	X =  1242.484  mm,	Y =   -38.517  mm,	Z =  2264.100  mm,
	W =   -32.017 deg,	P =   -31.509 deg,	R =    19.354 deg
   GP2:
	UF : 0, UT : 1,
	J1=   131.188 deg,	J2=   180.000 deg
};
P[910]{
   GP1:
	UF : 1, UT : 1,		CONFIG : 'N U T, 0, 0, 0',
	X =  1678.533  mm,	Y =  -253.828  mm,	Z =  2096.179  mm,
	W =   -44.666 deg,	P =    -5.995 deg,	R =    -2.790 deg
   GP2:
	UF : 0, UT : 1,
	J1=   131.188 deg,	J2=   180.000 deg
};
P[911]{
   GP1:
	UF : 1, UT : 1,		CONFIG : 'N U T, 0, 0, 0',
	X =  1703.320  mm,	Y =  -397.922  mm,	Z =  1954.333  mm,
	W =   -45.225 deg,	P =    -9.980 deg,	R =     1.224 deg
   GP2:
	UF : 0, UT : 1,
	J1=   131.188 deg,	J2=   180.000 deg
};
P[912]{
   GP1:
	UF : 1, UT : 1,		CONFIG : 'N U T, 0, 0, 0',
	X =  1675.864  mm,	Y =  -397.713  mm,	Z =  1947.138  mm,
	W =   -45.494 deg,	P =    11.391 deg,	R =   -20.046 deg
   GP2:
	UF : 0, UT : 1,
	J1=   131.188 deg,	J2=   180.000 deg
};
P[913]{
   GP1:
	UF : 1, UT : 1,		CONFIG : 'N U T, 0, 0, 0',
	X =  1728.670  mm,	Y =  -309.937  mm,	Z =  2044.029  mm,
	W =   -44.670 deg,	P =    -6.034 deg,	R =    -2.751 deg
   GP2:
	UF : 0, UT : 1,
	J1=   131.188 deg,	J2=   180.000 deg
};
P[914]{
   GP1:
	UF : 1, UT : 1,		CONFIG : 'N U T, 0, 0, 0',
	X =  1347.300  mm,	Y =  -220.973  mm,	Z =  2082.770  mm,
	W =    -1.262 deg,	P =   -15.279 deg,	R =     7.041 deg
   GP2:
	UF : 0, UT : 1,
	J1=   131.188 deg,	J2=   180.000 deg
};
P[915]{
   GP1:
	UF : 1, UT : 1,		CONFIG : 'N U T, 0, 0, 0',
	X =  1532.066  mm,	Y =  -519.406  mm,	Z =  1979.773  mm,
	W =    51.555 deg,	P =   -29.157 deg,	R =   -17.061 deg
   GP2:
	UF : 0, UT : 1,
	J1=   131.188 deg,	J2=   180.000 deg
};
P[916]{
   GP1:
	UF : 1, UT : 1,		CONFIG : 'N U T, 0, 0, 0',
	X =  1584.004  mm,	Y =  -453.419  mm,	Z =  1925.477  mm,
	W =    50.527 deg,	P =   -27.619 deg,	R =   -14.899 deg
   GP2:
	UF : 0, UT : 1,
	J1=   131.188 deg,	J2=   180.000 deg
};
P[917]{
   GP1:
	UF : 1, UT : 1,		CONFIG : 'N U T, 0, 0, 0',
	X =  1608.931  mm,	Y =  -453.588  mm,	Z =  1930.522  mm,
	W =    58.344 deg,	P =   -36.533 deg,	R =   -29.518 deg
   GP2:
	UF : 0, UT : 1,
	J1=   131.188 deg,	J2=   180.000 deg
};
P[918]{
   GP1:
	UF : 1, UT : 1,		CONFIG : 'N U T, 0, 0, 0',
	X =  1533.758  mm,	Y =  -508.845  mm,	Z =  1967.543  mm,
	W =    58.344 deg,	P =   -36.533 deg,	R =   -29.518 deg
   GP2:
	UF : 0, UT : 1,
	J1=   131.188 deg,	J2=   180.000 deg
};
P[919]{
   GP1:
	UF : 1, UT : 1,		CONFIG : 'N U T, 0, 0, 0',
	X =   982.914  mm,	Y =  -164.140  mm,	Z =  2330.780  mm,
	W =    27.111 deg,	P =   -49.789 deg,	R =    -8.012 deg
   GP2:
	UF : 0, UT : 1,
	J1=   131.201 deg,	J2=   180.000 deg
};
P[920]{
   GP1:
	UF : 1, UT : 1,		CONFIG : 'N U B, 0, 0, 0',
	X =   357.017  mm,	Y =     -.146  mm,	Z =  2433.121  mm,
	W =     -.021 deg,	P =   -39.773 deg,	R =      .020 deg
   GP2:
	UF : 0, UT : 1,
	J1=   180.000 deg,	J2=   180.000 deg
};
P[921]{
   GP1:
	UF : 1, UT : 1,
	J1=    22.718 deg,	J2=   -77.953 deg,	J3=    36.710 deg,
	J4=   -12.090 deg,	J5=  -103.365 deg,	J6=   138.265 deg
   GP2:
	UF : 0, UT : 1,
	J1=   180.000 deg,	J2=   180.000 deg
};
P[922]{
   GP1:
	UF : 1, UT : 1,		CONFIG : 'N U T, 0, 0, 0',
	X =   602.106  mm,	Y =   266.643  mm,	Z =   883.671  mm,
	W =   -17.511 deg,	P =    41.069 deg,	R =   154.352 deg
   GP2:
	UF : 0, UT : 1,
	J1=   180.000 deg,	J2=   180.000 deg
};
P[923]{
   GP1:
	UF : 1, UT : 1,		CONFIG : 'N U T, 0, 0, 0',
	X =   689.759  mm,	Y =   315.348  mm,	Z =   765.249  mm,
	W =   -18.279 deg,	P =    41.594 deg,	R =   154.204 deg
   GP2:
	UF : 0, UT : 1,
	J1=   179.999 deg,	J2=   180.000 deg
};
P[924]{
   GP1:
	UF : 1, UT : 1,		CONFIG : 'N U T, 0, 0, 0',
	X =   689.903  mm,	Y =   396.000  mm,	Z =   764.634  mm,
	W =   -33.904 deg,	P =    30.686 deg,	R =   141.051 deg
   GP2:
	UF : 0, UT : 1,
	J1=   179.999 deg,	J2=   180.000 deg
};
P[925]{
   GP1:
	UF : 1, UT : 1,		CONFIG : 'N U T, 0, 0, 0',
	X =   622.859  mm,	Y =   323.993  mm,	Z =   865.068  mm,
	W =   -39.588 deg,	P =    22.282 deg,	R =   128.236 deg
   GP2:
	UF : 0, UT : 1,
	J1=   180.000 deg,	J2=   180.000 deg
};
P[926]{
   GP1:
	UF : 1, UT : 1,		CONFIG : 'N U T, 0, 0, 0',
	X =   680.932  mm,	Y =   285.143  mm,	Z =   802.173  mm,
	W =   -39.374 deg,	P =    23.831 deg,	R =   116.224 deg
   GP2:
	UF : 0, UT : 1,
	J1=   180.000 deg,	J2=   180.000 deg
};
P[927]{
   GP1:
	UF : 1, UT : 1,		CONFIG : 'N U T, 0, 0, 0',
	X =   688.962  mm,	Y =   283.100  mm,	Z =   763.526  mm,
	W =   -39.397 deg,	P =    23.722 deg,	R =   115.040 deg
   GP2:
	UF : 0, UT : 1,
	J1=   180.000 deg,	J2=   180.000 deg
};
P[928]{
   GP1:
	UF : 1, UT : 1,		CONFIG : 'N U T, 0, 0, 1',
	X =   692.133  mm,	Y =  -280.944  mm,	Z =   761.510  mm,
	W =    -8.965 deg,	P =    44.205 deg,	R =   161.967 deg
   GP2:
	UF : 0, UT : 1,
	J1=   179.999 deg,	J2=   180.000 deg
};
P[929]{
   GP1:
	UF : 1, UT : 1,		CONFIG : 'N U T, 0, 0, 0',
	X =   629.190  mm,	Y =  -329.647  mm,	Z =   856.249  mm,
	W =    17.347 deg,	P =    49.328 deg,	R =   167.149 deg
   GP2:
	UF : 0, UT : 1,
	J1=   180.000 deg,	J2=   180.000 deg
};
P[930]{
   GP1:
	UF : 1, UT : 1,		CONFIG : 'N U T, 0, 0, 0',
	X =   623.987  mm,	Y =  -320.770  mm,	Z =   915.725  mm,
	W =   -33.842 deg,	P =    54.847 deg,	R =    56.315 deg
   GP2:
	UF : 0, UT : 1,
	J1=   180.000 deg,	J2=   180.000 deg
};
P[931]{
   GP1:
	UF : 1, UT : 1,		CONFIG : 'N U T, 0, 0, 0',
	X =   677.066  mm,	Y =  -284.917  mm,	Z =  1000.353  mm,
	W =    34.269 deg,	P =    57.953 deg,	R =  -154.245 deg
   GP2:
	UF : 0, UT : 1,
	J1=   180.000 deg,	J2=   180.000 deg
};
P[932]{
   GP1:
	UF : 1, UT : 1,		CONFIG : 'N U T, 0, 0, 0',
	X =   690.762  mm,	Y =  -320.058  mm,	Z =   764.207  mm,
	W =    35.931 deg,	P =    30.851 deg,	R =  -126.428 deg
   GP2:
	UF : 0, UT : 1,
	J1=   180.000 deg,	J2=   180.000 deg
};
P[933]{
   GP1:
	UF : 1, UT : 1,		CONFIG : 'N U T, 0, 0, 0',
	X =   688.887  mm,	Y =  -397.684  mm,	Z =   767.057  mm,
	W =    39.449 deg,	P =    23.626 deg,	R =  -129.170 deg
   GP2:
	UF : 0, UT : 1,
	J1=   179.999 deg,	J2=   180.000 deg
};
P[934]{
   GP1:
	UF : 1, UT : 1,		CONFIG : 'N U T, 0, 0, 1',
	X =   415.579  mm,	Y =  -304.795  mm,	Z =  1078.946  mm,
	W =    41.082 deg,	P =    20.266 deg,	R =  -127.997 deg
   GP2:
	UF : 0, UT : 1,
	J1=   180.000 deg,	J2=   180.000 deg
};
P[935]{
   GP1:
	UF : 1, UT : 1,
	J1=   -50.075 deg,	J2=   -70.188 deg,	J3=    26.322 deg,
	J4=   -22.185 deg,	J5=   -51.288 deg,	J6=    85.470 deg
   GP2:
	UF : 0, UT : 1,
	J1=   180.000 deg,	J2=   196.129 deg
};
P[936]{
   GP1:
	UF : 1, UT : 1,		CONFIG : 'N U T, 0, 0, 0',
	X =   917.635  mm,	Y =  -753.233  mm,	Z =  1083.148  mm,
	W =   -38.429 deg,	P =   -34.649 deg,	R =      .780 deg
   GP2:
	UF : 0, UT : 1,
	J1=   180.000 deg,	J2=   196.129 deg
};
P[937]{
   GP1:
	UF : 1, UT : 1,		CONFIG : 'N U T, 0, 0, 0',
	X =   931.634  mm,	Y =  -796.590  mm,	Z =  1036.018  mm,
	W =   -35.829 deg,	P =   -29.161 deg,	R =    -4.112 deg
   GP2:
	UF : 0, UT : 1,
	J1=   180.000 deg,	J2=   196.129 deg
};
P[938]{
   GP1:
	UF : 1, UT : 1,		CONFIG : 'N U T, 0, 0, 0',
	X =  1027.983  mm,	Y =  -767.049  mm,	Z =  1037.107  mm,
	W =   -37.222 deg,	P =   -35.147 deg,	R =     4.026 deg
   GP2:
	UF : 0, UT : 1,
	J1=   180.000 deg,	J2=   196.129 deg
};
P[939]{
   GP1:
	UF : 1, UT : 1,		CONFIG : 'N U T, 0, 0, 0',
	X =  1019.216  mm,	Y =  -755.446  mm,	Z =  1086.674  mm,
	W =   -73.601 deg,	P =   -18.162 deg,	R =    24.579 deg
   GP2:
	UF : 0, UT : 1,
	J1=   180.000 deg,	J2=   196.129 deg
};
P[940]{
   GP1:
	UF : 1, UT : 1,		CONFIG : 'N U T, 0, 0, 0',
	X =   651.216  mm,	Y =  -755.446  mm,	Z =  1093.416  mm,
	W =   -73.601 deg,	P =   -18.162 deg,	R =    24.579 deg
   GP2:
	UF : 0, UT : 1,
	J1=   180.000 deg,	J2=   196.129 deg
};
P[941]{
   GP1:
	UF : 1, UT : 1,		CONFIG : 'N U T, 0, 0, 0',
	X =   879.312  mm,	Y =  -733.458  mm,	Z =  1043.745  mm,
	W =     -.609 deg,	P =   -11.317 deg,	R =    19.232 deg
   GP2:
	UF : 0, UT : 1,
	J1=   180.000 deg,	J2=   196.129 deg
};
P[942]{
   GP1:
	UF : 1, UT : 1,		CONFIG : 'N U T, 0, 0, 0',
	X =   879.754  mm,	Y =  -733.151  mm,	Z =   977.386  mm,
	W =    -3.361 deg,	P =   -10.118 deg,	R =    19.733 deg
   GP2:
	UF : 0, UT : 1,
	J1=   180.000 deg,	J2=   196.129 deg
};
P[943]{
   GP1:
	UF : 1, UT : 1,		CONFIG : 'N U T, 0, 0, 0',
	X =   895.508  mm,	Y =  -786.854  mm,	Z =   973.466  mm,
	W =   -11.891 deg,	P =      .117 deg,	R =    18.403 deg
   GP2:
	UF : 0, UT : 1,
	J1=   180.000 deg,	J2=   196.129 deg
};
P[944]{
   GP1:
	UF : 1, UT : 1,		CONFIG : 'N U T, 0, 0, 0',
	X =   894.892  mm,	Y =  -773.751  mm,	Z =  1072.111  mm,
	W =   -11.972 deg,	P =    -6.765 deg,	R =    19.858 deg
   GP2:
	UF : 0, UT : 1,
	J1=   180.000 deg,	J2=   196.129 deg
};
P[945]{
   GP1:
	UF : 1, UT : 1,		CONFIG : 'N U T, 0, 0, 0',
	X =   796.225  mm,	Y =  -784.763  mm,	Z =  1290.070  mm,
	W =   -16.270 deg,	P =     1.406 deg,	R =    16.682 deg
   GP2:
	UF : 0, UT : 1,
	J1=   180.000 deg,	J2=   196.129 deg
};
P[946]{
   GP1:
	UF : 1, UT : 1,		CONFIG : 'N U T, 0, 0, 0',
	X =   455.144  mm,	Y =  -223.806  mm,	Z =  1838.943  mm,
	W =  -100.113 deg,	P =   -16.084 deg,	R =    32.515 deg
   GP2:
	UF : 0, UT : 1,
	J1=   180.000 deg,	J2=   196.129 deg
};
P[947]{
   GP1:
	UF : 1, UT : 1,		CONFIG : 'N U T, 0, 0, 0',
	X =   433.199  mm,	Y =   723.768  mm,	Z =  1735.241  mm,
	W =    31.808 deg,	P =   -58.935 deg,	R =    27.008 deg
   GP2:
	UF : 0, UT : 1,
	J1=   180.000 deg,	J2=   162.834 deg
};
P[948]{
   GP1:
	UF : 1, UT : 1,		CONFIG : 'N U T, 0, 0, 0',
	X =   915.388  mm,	Y =   803.489  mm,	Z =  1076.813  mm,
	W =    31.157 deg,	P =   -41.097 deg,	R =    13.870 deg
   GP2:
	UF : 0, UT : 1,
	J1=   180.000 deg,	J2=   162.834 deg
};
P[949]{
   GP1:
	UF : 1, UT : 1,		CONFIG : 'N U T, 0, 0, 0',
	X =   945.882  mm,	Y =   822.490  mm,	Z =  1036.624  mm,
	W =    31.211 deg,	P =   -41.079 deg,	R =    13.849 deg
   GP2:
	UF : 0, UT : 1,
	J1=   180.000 deg,	J2=   162.834 deg
};
P[950]{
   GP1:
	UF : 1, UT : 1,		CONFIG : 'N U T, 0, 0, 0',
	X =  1045.978  mm,	Y =   792.926  mm,	Z =  1034.331  mm,
	W =    32.243 deg,	P =   -40.608 deg,	R =    13.275 deg
   GP2:
	UF : 0, UT : 1,
	J1=   179.999 deg,	J2=   162.834 deg
};
P[951]{
   GP1:
	UF : 1, UT : 1,		CONFIG : 'N U T, 0, 0, 0',
	X =  1039.367  mm,	Y =   769.241  mm,	Z =  1064.643  mm,
	W =    35.123 deg,	P =   -46.989 deg,	R =     8.148 deg
   GP2:
	UF : 0, UT : 1,
	J1=   180.000 deg,	J2=   162.834 deg
};
P[952]{
   GP1:
	UF : 1, UT : 1,		CONFIG : 'N U T, 0, 0, 0',
	X =   869.380  mm,	Y =   769.192  mm,	Z =  1065.308  mm,
	W =    35.418 deg,	P =   -46.890 deg,	R =     7.970 deg
   GP2:
	UF : 0, UT : 1,
	J1=   179.999 deg,	J2=   162.834 deg
};
P[953]{
   GP1:
	UF : 1, UT : 1,		CONFIG : 'N U T, 0, 0, 0',
	X =   861.004  mm,	Y =   762.759  mm,	Z =  1052.130  mm,
	W =    -7.907 deg,	P =    -8.124 deg,	R =    27.444 deg
   GP2:
	UF : 0, UT : 1,
	J1=   180.000 deg,	J2=   162.834 deg
};
P[954]{
   GP1:
	UF : 1, UT : 1,		CONFIG : 'N U T, 0, 0, 0',
	X =   895.848  mm,	Y =   757.903  mm,	Z =   977.410  mm,
	W =    -6.316 deg,	P =    -5.173 deg,	R =    27.290 deg
   GP2:
	UF : 0, UT : 1,
	J1=   180.000 deg,	J2=   162.834 deg
};
P[955]{
   GP1:
	UF : 1, UT : 1,		CONFIG : 'N U T, 0, 0, 0',
	X =   911.616  mm,	Y =   812.935  mm,	Z =   977.333  mm,
	W =    -5.644 deg,	P =    -3.900 deg,	R =    27.238 deg
   GP2:
	UF : 0, UT : 1,
	J1=   180.000 deg,	J2=   162.834 deg
};
P[956]{
   GP1:
	UF : 1, UT : 1,		CONFIG : 'N U T, 0, 0, 0',
	X =   915.146  mm,	Y =   811.304  mm,	Z =  1045.569  mm,
	W =     -.314 deg,	P =    -5.430 deg,	R =    27.373 deg
   GP2:
	UF : 0, UT : 1,
	J1=   180.000 deg,	J2=   162.834 deg
};
P[957]{
   GP1:
	UF : 1, UT : 1,		CONFIG : 'N U T, 0, 0, 0',
	X =   697.391  mm,	Y =   811.304  mm,	Z =  1325.569  mm,
	W =     -.314 deg,	P =    -5.430 deg,	R =    27.373 deg
   GP2:
	UF : 0, UT : 1,
	J1=   180.000 deg,	J2=   162.834 deg
};
P[958]{
   GP1:
	UF : 1, UT : 1,		CONFIG : 'N U B, 0, 0, 0',
	X =   357.017  mm,	Y =     -.146  mm,	Z =  2433.121  mm,
	W =     -.021 deg,	P =   -39.773 deg,	R =      .020 deg
   GP2:
	UF : 0, UT : 1,
	J1=   180.000 deg,	J2=   162.834 deg
};
P[959]{
   GP1:
	UF : 1, UT : 1,		CONFIG : 'N U B, 0, 0, 0',
	X =   357.017  mm,	Y =     -.146  mm,	Z =  2433.121  mm,
	W =     -.021 deg,	P =   -39.773 deg,	R =      .020 deg
   GP2:
	UF : 0, UT : 1,
	J1=    90.000 deg,	J2=   180.000 deg
};
P[960]{
   GP1:
	UF : 1, UT : 1,		CONFIG : 'N U T, 0, 0, 0',
	X =  2079.740  mm,	Y =     2.655  mm,	Z =  1634.851  mm,
	W =   -39.435 deg,	P =    38.877 deg,	R =    63.496 deg
   GP2:
	UF : 0, UT : 1,
	J1=    90.000 deg,	J2=   180.000 deg
};
P[961]{
   GP1:
	UF : 1, UT : 1,		CONFIG : 'N U T, 0, 0, 0',
	X =  2641.070  mm,	Y =    96.952  mm,	Z =   892.786  mm,
	W =   -30.662 deg,	P =    38.178 deg,	R =    67.355 deg
   GP2:
	UF : 0, UT : 1,
	J1=    90.000 deg,	J2=   180.000 deg
};
P[962]{
   GP1:
	UF : 1, UT : 1,		CONFIG : 'N U T, 0, 0, 0',
	X =  2779.073  mm,	Y =    63.988  mm,	Z =   854.225  mm,
	W =   -27.596 deg,	P =    28.973 deg,	R =    42.829 deg
   GP2:
	UF : 0, UT : 1,
	J1=    90.000 deg,	J2=   180.000 deg
};
P[963]{
   GP1:
	UF : 1, UT : 1,		CONFIG : 'N U T, 0, 0, 0',
	X =  2793.089  mm,	Y =    50.841  mm,	Z =   752.992  mm,
	W =   -32.482 deg,	P =    32.696 deg,	R =    40.318 deg
   GP2:
	UF : 0, UT : 1,
	J1=    90.000 deg,	J2=   180.000 deg
};
P[964]{
   GP1:
	UF : 1, UT : 1,		CONFIG : 'N U T, 0, 0, 0',
	X =  2827.763  mm,	Y =    50.645  mm,	Z =   753.413  mm,
	W =   -32.638 deg,	P =    32.806 deg,	R =    40.233 deg
   GP2:
	UF : 0, UT : 1,
	J1=    90.000 deg,	J2=   180.000 deg
};
P[965]{
   GP1:
	UF : 1, UT : 1,		CONFIG : 'N U T, 0, 0, 0',
	X =  2793.338  mm,	Y =    82.464  mm,	Z =   838.649  mm,
	W =   -26.653 deg,	P =    28.198 deg,	R =    43.280 deg
   GP2:
	UF : 0, UT : 1,
	J1=    90.000 deg,	J2=   180.000 deg
};
P[966]{
   GP1:
	UF : 1, UT : 1,		CONFIG : 'N U T, 0, 0, 0',
	X =  2807.102  mm,	Y =   -36.017  mm,	Z =   825.713  mm,
	W =    15.607 deg,	P =    10.488 deg,	R =   -33.094 deg
   GP2:
	UF : 0, UT : 1,
	J1=    90.000 deg,	J2=   180.000 deg
};
P[967]{
   GP1:
	UF : 1, UT : 1,		CONFIG : 'N U T, 0, 0, 0',
	X =  2792.338  mm,	Y =   -78.536  mm,	Z =   812.201  mm,
	W =    22.126 deg,	P =    31.326 deg,	R =   -51.965 deg
   GP2:
	UF : 0, UT : 1,
	J1=    90.000 deg,	J2=   180.000 deg
};
P[968]{
   GP1:
	UF : 1, UT : 1,		CONFIG : 'N U T, 0, 0, 0',
	X =  2799.457  mm,	Y =   -51.911  mm,	Z =   752.825  mm,
	W =    18.868 deg,	P =    36.472 deg,	R =   -60.103 deg
   GP2:
	UF : 0, UT : 1,
	J1=    90.000 deg,	J2=   180.000 deg
};
P[969]{
   GP1:
	UF : 1, UT : 1,		CONFIG : 'N U T, 0, 0, 0',
	X =  2829.014  mm,	Y =   -52.533  mm,	Z =   753.514  mm,
	W =    17.562 deg,	P =    37.061 deg,	R =   -62.294 deg
   GP2:
	UF : 0, UT : 1,
	J1=    90.000 deg,	J2=   180.000 deg
};
P[970]{
   GP1:
	UF : 1, UT : 1,		CONFIG : 'N U T, 0, 0, 0',
	X =  2792.338  mm,	Y =   -78.536  mm,	Z =   870.200  mm,
	W =    23.118 deg,	P =    32.394 deg,	R =   -51.441 deg
   GP2:
	UF : 0, UT : 1,
	J1=    90.000 deg,	J2=   180.000 deg
};
P[971]{
   GP1:
	UF : 1, UT : 1,		CONFIG : 'N U T, 0, 0, 0',
	X =  2792.338  mm,	Y =   -78.536  mm,	Z =   870.200  mm,
	W =     -.000 deg,	P =     6.847 deg,	R =      .007 deg
   GP2:
	UF : 0, UT : 1,
	J1=    90.000 deg,	J2=   180.000 deg
};
P[972]{
   GP1:
	UF : 1, UT : 1,		CONFIG : 'N U T, 0, 0, 0',
	X =  2852.717  mm,	Y =   -56.939  mm,	Z =   805.419  mm,
	W =      .000 deg,	P =    10.475 deg,	R =      .007 deg
   GP2:
	UF : 0, UT : 1,
	J1=    90.000 deg,	J2=   180.000 deg
};
P[973]{
   GP1:
	UF : 1, UT : 1,		CONFIG : 'N U T, 0, 0, 0',
	X =  2836.712  mm,	Y =   -51.940  mm,	Z =   754.621  mm,
	W =      .005 deg,	P =    15.556 deg,	R =      .002 deg
   GP2:
	UF : 0, UT : 1,
	J1=    90.000 deg,	J2=   180.000 deg
};
P[974]{
   GP1:
	UF : 1, UT : 1,		CONFIG : 'N U T, 0, 0, 0',
	X =  2837.937  mm,	Y =    51.593  mm,	Z =   753.607  mm,
	W =     -.000 deg,	P =    14.988 deg,	R =      .007 deg
   GP2:
	UF : 0, UT : 1,
	J1=    90.000 deg,	J2=   180.000 deg
};
P[975]{
   GP1:
	UF : 1, UT : 1,		CONFIG : 'N U T, 0, 0, 0',
	X =  2852.717  mm,	Y =   -56.939  mm,	Z =   805.419  mm,
	W =      .000 deg,	P =    10.475 deg,	R =      .007 deg
   GP2:
	UF : 0, UT : 1,
	J1=    90.000 deg,	J2=   180.000 deg
};
P[976]{
   GP1:
	UF : 1, UT : 1,		CONFIG : 'N U T, 0, 0, 0',
	X =  2698.431  mm,	Y =   -56.939  mm,	Z =  1002.562  mm,
	W =     -.002 deg,	P =   -13.112 deg,	R =      .007 deg
   GP2:
	UF : 0, UT : 1,
	J1=    90.000 deg,	J2=   180.000 deg
};
P[977]{
   GP1:
	UF : 1, UT : 1,		CONFIG : 'N U T, 0, 0, 0',
	X =  1186.431  mm,	Y =   -56.939  mm,	Z =  1002.561  mm,
	W =     -.002 deg,	P =   -13.112 deg,	R =      .007 deg
   GP2:
	UF : 0, UT : 1,
	J1=    90.000 deg,	J2=   180.000 deg
};
P[978]{
   GP1:
	UF : 1, UT : 1,		CONFIG : 'N U T, 0, 0, 0',
	X =  1422.321  mm,	Y =   -19.612  mm,	Z =   892.933  mm,
	W =      .000 deg,	P =    43.571 deg,	R =      .007 deg
   GP2:
	UF : 0, UT : 1,
	J1=    90.000 deg,	J2=   180.000 deg
};
P[979]{
   GP1:
	UF : 1, UT : 1,		CONFIG : 'N U T, 0, 0, 0',
	X =  1709.321  mm,	Y =  -382.612  mm,	Z =   539.934  mm,
	W =     0.000 deg,	P =    43.571 deg,	R =    90.007 deg
   GP2:
	UF : 0, UT : 1,
	J1=    90.000 deg,	J2=   180.000 deg
};
P[980]{
   GP1:
	UF : 1, UT : 1,		CONFIG : 'N U T, 0, 0, 0',
	X =  1716.341  mm,	Y =  -449.493  mm,	Z =   422.245  mm,
	W =     -.012 deg,	P =    43.506 deg,	R =    86.332 deg
   GP2:
	UF : 1, UT : 1,
	J1=    90.000 deg,	J2=   180.000 deg
};
P[981]{
   GP1:
	UF : 1, UT : 1,		CONFIG : 'N U T, 0, 0, 0',
	X =  1584.270  mm,	Y =  -447.721  mm,	Z =   422.331  mm,
	W =     -.013 deg,	P =    43.517 deg,	R =    86.261 deg
   GP2:
	UF : 1, UT : 1,
	J1=    90.000 deg,	J2=   180.000 deg
};
P[982]{
   GP1:
	UF : 1, UT : 1,		CONFIG : 'N U T, 0, 0, 0',
	X =  1599.753  mm,	Y =  -381.366  mm,	Z =   505.008  mm,
	W =      .000 deg,	P =    43.571 deg,	R =    86.288 deg
   GP2:
	UF : 0, UT : 1,
	J1=    90.000 deg,	J2=   180.000 deg
};
P[983]{
   GP1:
	UF : 1, UT : 1,		CONFIG : 'N U T, 0, 0, 0',
	X =  1999.753  mm,	Y =  -381.366  mm,	Z =   505.007  mm,
	W =   -38.646 deg,	P =    21.930 deg,	R =    21.323 deg
   GP2:
	UF : 0, UT : 1,
	J1=    90.000 deg,	J2=   180.000 deg
};
P[984]{
   GP1:
	UF : 1, UT : 1,		CONFIG : 'N U T, 0, 0, 0',
	X =  1957.623  mm,	Y =  -442.508  mm,	Z =   427.694  mm,
	W =   -40.830 deg,	P =    20.791 deg,	R =    22.336 deg
   GP2:
	UF : 1, UT : 1,
	J1=    90.000 deg,	J2=   180.000 deg
};
P[985]{
   GP1:
	UF : 1, UT : 1,		CONFIG : 'N U T, 0, 0, 0',
	X =  2028.883  mm,	Y =  -449.653  mm,	Z =   423.872  mm,
	W =   -42.077 deg,	P =    21.682 deg,	R =    36.466 deg
   GP2:
	UF : 1, UT : 1,
	J1=    90.000 deg,	J2=   180.000 deg
};
P[986]{
   GP1:
	UF : 1, UT : 1,		CONFIG : 'N U T, 0, 0, 0',
	X =  2048.708  mm,	Y =  -116.976  mm,	Z =   584.258  mm,
	W =   -38.646 deg,	P =    21.930 deg,	R =    21.323 deg
   GP2:
	UF : 0, UT : 1,
	J1=    90.000 deg,	J2=   180.000 deg
};
P[987]{
   GP1:
	UF : 1, UT : 1,		CONFIG : 'N U T, 0, 0, 0',
	X =  2054.995  mm,	Y =  -300.976  mm,	Z =   557.316  mm,
	W =   -43.351 deg,	P =    -4.892 deg,	R =    40.339 deg
   GP2:
	UF : 0, UT : 1,
	J1=    90.000 deg,	J2=   180.000 deg
};
P[988]{
   GP1:
	UF : 1, UT : 1,		CONFIG : 'N U T, 0, 0, 0',
	X =  2146.567  mm,	Y =  -386.362  mm,	Z =   419.052  mm,
	W =   -44.859 deg,	P =    -3.606 deg,	R =    27.054 deg
   GP2:
	UF : 1, UT : 1,
	J1=    90.000 deg,	J2=   180.000 deg
};
P[989]{
   GP1:
	UF : 1, UT : 1,		CONFIG : 'N U T, 0, 0, 0',
	X =  2105.985  mm,	Y =  -419.849  mm,	Z =   419.949  mm,
	W =   -43.242 deg,	P =    13.881 deg,	R =    57.005 deg
   GP2:
	UF : 1, UT : 1,
	J1=    90.000 deg,	J2=   180.000 deg
};
P[990]{
   GP1:
	UF : 1, UT : 1,		CONFIG : 'N U T, 0, 0, 0',
	X =  2099.851  mm,	Y =  -426.411  mm,	Z =   422.441  mm,
	W =   -43.579 deg,	P =    -9.861 deg,	R =    55.520 deg
   GP2:
	UF : 1, UT : 1,
	J1=    89.999 deg,	J2=   180.000 deg
};
P[991]{
   GP1:
	UF : 1, UT : 1,		CONFIG : 'N U T, 0, 0, 0',
	X =  2097.549  mm,	Y =  -435.485  mm,	Z =   422.872  mm,
	W =   -43.572 deg,	P =    -9.889 deg,	R =    55.498 deg
   GP2:
	UF : 1, UT : 1,
	J1=    89.999 deg,	J2=   180.000 deg
};
P[992]{
   GP1:
	UF : 1, UT : 1,		CONFIG : 'N U T, 0, 0, 0',
	X =  1981.542  mm,	Y =  -402.485  mm,	Z =   562.968  mm,
	W =   -43.468 deg,	P =    -3.333 deg,	R =    66.484 deg
   GP2:
	UF : 0, UT : 1,
	J1=    90.000 deg,	J2=   180.000 deg
};
P[993]{
   GP1:
	UF : 1, UT : 1,		CONFIG : 'N U T, 0, 0, 0',
	X =  1422.321  mm,	Y =   -19.612  mm,	Z =   902.933  mm,
	W =      .000 deg,	P =    43.571 deg,	R =      .007 deg
   GP2:
	UF : 0, UT : 1,
	J1=    90.000 deg,	J2=   180.000 deg
};
P[994]{
   GP1:
	UF : 1, UT : 1,		CONFIG : 'N U T, 0, 0, 0',
	X =  1722.321  mm,	Y =   380.388  mm,	Z =   483.934  mm,
	W =     0.000 deg,	P =    43.571 deg,	R =   -89.993 deg
   GP2:
	UF : 0, UT : 1,
	J1=    90.000 deg,	J2=   180.000 deg
};
P[995]{
   GP1:
	UF : 1, UT : 1,		CONFIG : 'N U T, 0, 0, 0',
	X =  1718.837  mm,	Y =   444.280  mm,	Z =   423.719  mm,
	W =    -1.652 deg,	P =    44.986 deg,	R =   -90.065 deg
   GP2:
	UF : 1, UT : 1,
	J1=    90.000 deg,	J2=   180.000 deg
};
P[996]{
   GP1:
	UF : 1, UT : 1,		CONFIG : 'N U T, 0, 0, 0',
	X =  1588.480  mm,	Y =   444.279  mm,	Z =   420.719  mm,
	W =    -1.652 deg,	P =    44.986 deg,	R =   -90.065 deg
   GP2:
	UF : 1, UT : 1,
	J1=    90.000 deg,	J2=   180.000 deg
};
P[997]{
   GP1:
	UF : 1, UT : 1,		CONFIG : 'N U T, 0, 0, 0',
	X =  1595.927  mm,	Y =   343.841  mm,	Z =   518.086  mm,
	W =      .000 deg,	P =    43.571 deg,	R =   -92.306 deg
   GP2:
	UF : 0, UT : 1,
	J1=    90.000 deg,	J2=   180.000 deg
};
P[998]{
   GP1:
	UF : 1, UT : 1,		CONFIG : 'N U T, 0, 0, 0',
	X =  1973.927  mm,	Y =   343.841  mm,	Z =   518.086  mm,
	W =    31.879 deg,	P =    31.438 deg,	R =   -42.291 deg
   GP2:
	UF : 0, UT : 1,
	J1=    90.000 deg,	J2=   180.000 deg
};
P[999]{
   GP1:
	UF : 1, UT : 1,		CONFIG : 'N U T, 0, 0, 0',
	X =  1958.374  mm,	Y =   445.827  mm,	Z =   422.299  mm,
	W =    32.302 deg,	P =    33.270 deg,	R =   -47.081 deg
   GP2:
	UF : 1, UT : 1,
	J1=    90.000 deg,	J2=   180.000 deg
};
P[1000]{
   GP1:
	UF : 1, UT : 1,		CONFIG : 'N U T, 0, 0, 0',
	X =  2032.108  mm,	Y =   448.090  mm,	Z =   422.222  mm,
	W =    43.758 deg,	P =    22.369 deg,	R =   -31.690 deg
   GP2:
	UF : 1, UT : 1,
	J1=    90.000 deg,	J2=   180.000 deg
};
P[1001]{
   GP1:
	UF : 1, UT : 1,		CONFIG : 'N U T, 0, 0, 0',
	X =  2029.632  mm,	Y =   298.067  mm,	Z =   568.513  mm,
	W =    39.948 deg,	P =    19.080 deg,	R =   -23.626 deg
   GP2:
	UF : 0, UT : 1,
	J1=    90.000 deg,	J2=   180.000 deg
};
P[1002]{
   GP1:
	UF : 1, UT : 1,		CONFIG : 'N U T, 0, 0, 0',
	X =  2029.631  mm,	Y =   298.067  mm,	Z =   568.513  mm,
	W =    39.948 deg,	P =    19.080 deg,	R =   -73.748 deg
   GP2:
	UF : 0, UT : 1,
	J1=    90.000 deg,	J2=   180.000 deg
};
P[1003]{
   GP1:
	UF : 1, UT : 1,		CONFIG : 'N U T, 0, 0, 0',
	X =  2146.180  mm,	Y =   383.228  mm,	Z =   419.895  mm,
	W =    42.404 deg,	P =    16.917 deg,	R =   -60.322 deg
   GP2:
	UF : 1, UT : 1,
	J1=    90.000 deg,	J2=   180.000 deg
};
P[1004]{
   GP1:
	UF : 1, UT : 1,		CONFIG : 'N U T, 0, 0, 0',
	X =  2105.246  mm,	Y =   421.815  mm,	Z =   420.684  mm,
	W =    44.162 deg,	P =     9.896 deg,	R =   -52.694 deg
   GP2:
	UF : 1, UT : 1,
	J1=    90.000 deg,	J2=   180.000 deg
};
P[1005]{
   GP1:
	UF : 1, UT : 1,		CONFIG : 'N U T, 0, 0, 0',
	X =  2102.134  mm,	Y =   425.996  mm,	Z =   421.012  mm,
	W =    44.143 deg,	P =     9.905 deg,	R =   -66.074 deg
   GP2:
	UF : 1, UT : 1,
	J1=    90.000 deg,	J2=   180.000 deg
};
P[1006]{
   GP1:
	UF : 1, UT : 1,		CONFIG : 'N U T, 0, 0, 0',
	X =  2100.705  mm,	Y =   433.132  mm,	Z =   421.964  mm,
	W =    44.953 deg,	P =     2.229 deg,	R =   -67.460 deg
   GP2:
	UF : 1, UT : 1,
	J1=    90.000 deg,	J2=   180.000 deg
};
P[1007]{
   GP1:
	UF : 1, UT : 1,		CONFIG : 'N U T, 0, 0, 0',
	X =  2003.428  mm,	Y =   126.931  mm,	Z =   541.830  mm,
	W =    43.132 deg,	P =    -6.887 deg,	R =   -61.237 deg
   GP2:
	UF : 0, UT : 1,
	J1=    90.000 deg,	J2=   180.000 deg
};
P[1008]{
   GP1:
	UF : 1, UT : 1,		CONFIG : 'N U T, 0, 0, 0',
	X =  2378.427  mm,	Y =   231.931  mm,	Z =   285.830  mm,
	W =    40.241 deg,	P =    18.349 deg,	R =   -20.268 deg
   GP2:
	UF : 0, UT : 1,
	J1=    90.000 deg,	J2=   180.000 deg
};
P[1009]{
   GP1:
	UF : 1, UT : 1,		CONFIG : 'N U T, 0, 0, 0',
	X =  2356.954  mm,	Y =   365.993  mm,	Z =   296.590  mm,
	W =    40.241 deg,	P =    18.349 deg,	R =   -20.268 deg
   GP2:
	UF : 0, UT : 1,
	J1=    90.000 deg,	J2=   180.000 deg
};
P[1010]{
   GP1:
	UF : 1, UT : 1,		CONFIG : 'N U T, 0, 0, 0',
	X =  2347.760  mm,	Y =   439.275  mm,	Z =   270.025  mm,
	W =    43.558 deg,	P =    12.622 deg,	R =   -12.919 deg
   GP2:
	UF : 0, UT : 1,
	J1=    90.000 deg,	J2=   180.000 deg
};
P[1011]{
   GP1:
	UF : 1, UT : 1,		CONFIG : 'N U T, 0, 0, 0',
	X =  2403.053  mm,	Y =   435.363  mm,	Z =   273.433  mm,
	W =    43.549 deg,	P =     1.536 deg,	R =   -16.674 deg
   GP2:
	UF : 0, UT : 1,
	J1=    90.000 deg,	J2=   180.000 deg
};
P[1012]{
   GP1:
	UF : 1, UT : 1,		CONFIG : 'N U T, 0, 0, 0',
	X =  2356.954  mm,	Y =   365.993  mm,	Z =   296.590  mm,
	W =    40.241 deg,	P =    18.349 deg,	R =   -20.268 deg
   GP2:
	UF : 0, UT : 1,
	J1=    90.000 deg,	J2=   180.000 deg
};
P[1013]{
   GP1:
	UF : 1, UT : 1,		CONFIG : 'N U T, 0, 0, 0',
	X =  2356.954  mm,	Y =   213.993  mm,	Z =   296.590  mm,
	W =    40.242 deg,	P =    18.350 deg,	R =   -20.267 deg
   GP2:
	UF : 0, UT : 1,
	J1=    90.000 deg,	J2=   180.000 deg
};
P[1014]{
   GP1:
	UF : 1, UT : 1,		CONFIG : 'N U T, 0, 0, 0',
	X =  2485.906  mm,	Y =   213.993  mm,	Z =   296.590  mm,
	W =    43.394 deg,	P =    -4.399 deg,	R =     4.775 deg
   GP2:
	UF : 0, UT : 1,
	J1=    90.000 deg,	J2=   180.000 deg
};
P[1015]{
   GP1:
	UF : 1, UT : 1,		CONFIG : 'N U T, 0, 0, 0',
	X =  2485.594  mm,	Y =   388.028  mm,	Z =   236.817  mm,
	W =    26.387 deg,	P =   -37.359 deg,	R =    50.769 deg
   GP2:
	UF : 0, UT : 1,
	J1=    90.000 deg,	J2=   180.000 deg
};
P[1016]{
   GP1:
	UF : 1, UT : 1,		CONFIG : 'N U T, 0, 0, 0',
	X =  2479.365  mm,	Y =   435.513  mm,	Z =   221.232  mm,
	W =    26.386 deg,	P =   -37.358 deg,	R =    60.941 deg
   GP2:
	UF : 0, UT : 1,
	J1=    90.000 deg,	J2=   180.000 deg
};
P[1017]{
   GP1:
	UF : 1, UT : 1,		CONFIG : 'N U T, 0, 0, 0',
	X =  2428.881  mm,	Y =   435.920  mm,	Z =   222.314  mm,
	W =    41.283 deg,	P =   -34.943 deg,	R =    58.712 deg
   GP2:
	UF : 0, UT : 1,
	J1=    90.000 deg,	J2=   180.000 deg
};
P[1018]{
   GP1:
	UF : 1, UT : 1,		CONFIG : 'N U T, 0, 0, 0',
	X =  2485.906  mm,	Y =   276.993  mm,	Z =   252.842  mm,
	W =    51.836 deg,	P =   -13.420 deg,	R =    11.542 deg
   GP2:
	UF : 0, UT : 1,
	J1=    90.000 deg,	J2=   180.000 deg
};
P[1019]{
   GP1:
	UF : 1, UT : 1,		CONFIG : 'N U T, 0, 0, 0',
	X =  2485.906  mm,	Y =   213.993  mm,	Z =   296.590  mm,
	W =    43.394 deg,	P =    -4.399 deg,	R =     4.775 deg
   GP2:
	UF : 0, UT : 1,
	J1=    90.000 deg,	J2=   180.000 deg
};
P[1020]{
   GP1:
	UF : 1, UT : 1,		CONFIG : 'N U T, 0, 0, 0',
	X =  2356.954  mm,	Y =    -6.007  mm,	Z =   296.591  mm,
	W =     5.759 deg,	P =    43.266 deg,	R =    98.508 deg
   GP2:
	UF : 0, UT : 1,
	J1=    90.000 deg,	J2=   180.000 deg
};
P[1021]{
   GP1:
	UF : 1, UT : 1,		CONFIG : 'N U T, 0, 0, 0',
	X =  2356.954  mm,	Y =  -371.775  mm,	Z =   296.590  mm,
	W =   -43.559 deg,	P =     1.197 deg,	R =     1.395 deg
   GP2:
	UF : 0, UT : 1,
	J1=    90.000 deg,	J2=   180.000 deg
};
P[1022]{
   GP1:
	UF : 1, UT : 1,		CONFIG : 'N U T, 0, 0, 0',
	X =  2348.791  mm,	Y =  -441.873  mm,	Z =   270.797  mm,
	W =   -44.984 deg,	P =     1.297 deg,	R =     5.834 deg
   GP2:
	UF : 0, UT : 1,
	J1=    90.000 deg,	J2=   180.000 deg
};
P[1023]{
   GP1:
	UF : 1, UT : 1,		CONFIG : 'N U T, 0, 0, 0',
	X =  2402.559  mm,	Y =  -440.035  mm,	Z =   275.286  mm,
	W =   -43.855 deg,	P =   -10.820 deg,	R =     5.503 deg
   GP2:
	UF : 0, UT : 1,
	J1=    90.000 deg,	J2=   180.000 deg
};
P[1024]{
   GP1:
	UF : 1, UT : 1,		CONFIG : 'N U T, 0, 0, 0',
	X =  2356.954  mm,	Y =  -368.775  mm,	Z =   284.590  mm,
	W =   -43.559 deg,	P =     1.197 deg,	R =     1.395 deg
   GP2:
	UF : 0, UT : 1,
	J1=    90.000 deg,	J2=   180.000 deg
};
P[1025]{
   GP1:
	UF : 1, UT : 1,		CONFIG : 'N U T, 0, 0, 0',
	X =  2356.954  mm,	Y =  -231.775  mm,	Z =   284.590  mm,
	W =   -43.560 deg,	P =     1.197 deg,	R =     1.395 deg
   GP2:
	UF : 0, UT : 1,
	J1=    90.000 deg,	J2=   180.000 deg
};
P[1026]{
   GP1:
	UF : 1, UT : 1,		CONFIG : 'N U T, 0, 0, 0',
	X =  2476.792  mm,	Y =  -231.775  mm,	Z =   284.590  mm,
	W =   -29.446 deg,	P =   -33.698 deg,	R =   -44.366 deg
   GP2:
	UF : 0, UT : 1,
	J1=    90.000 deg,	J2=   180.000 deg
};
P[1027]{
   GP1:
	UF : 1, UT : 1,		CONFIG : 'N U T, 0, 0, 0',
	X =  2481.972  mm,	Y =  -442.010  mm,	Z =   222.427  mm,
	W =    -2.397 deg,	P =   -44.949 deg,	R =   -86.609 deg
   GP2:
	UF : 0, UT : 1,
	J1=    90.000 deg,	J2=   180.000 deg
};
P[1028]{
   GP1:
	UF : 1, UT : 1,		CONFIG : 'N U T, 0, 0, 0',
	X =  2432.833  mm,	Y =  -441.320  mm,	Z =   222.622  mm,
	W =   -26.143 deg,	P =   -43.613 deg,	R =   -81.145 deg
   GP2:
	UF : 0, UT : 1,
	J1=    90.000 deg,	J2=   180.000 deg
};
P[1029]{
   GP1:
	UF : 1, UT : 1,		CONFIG : 'N U T, 0, 0, 0',
	X =  2488.923  mm,	Y =  -351.753  mm,	Z =   247.956  mm,
	W =   -30.826 deg,	P =   -42.294 deg,	R =   -63.160 deg
   GP2:
	UF : 0, UT : 1,
	J1=    90.000 deg,	J2=   180.000 deg
};
P[1030]{
   GP1:
	UF : 1, UT : 1,		CONFIG : 'N U T, 0, 0, 0',
	X =  2476.792  mm,	Y =  -231.776  mm,	Z =   284.590  mm,
	W =   -29.446 deg,	P =   -33.698 deg,	R =   -44.366 deg
   GP2:
	UF : 0, UT : 1,
	J1=    90.000 deg,	J2=   180.000 deg
};
P[1031]{
   GP1:
	UF : 1, UT : 1,		CONFIG : 'N U T, 0, 0, 0',
	X =  2405.334  mm,	Y =  -139.398  mm,	Z =   301.608  mm,
	W =   -39.075 deg,	P =    20.318 deg,	R =    23.103 deg
   GP2:
	UF : 0, UT : 1,
	J1=    90.000 deg,	J2=   180.000 deg
};
P[1032]{
   GP1:
	UF : 1, UT : 1,		CONFIG : 'N U B, 0, 0, 0',
	X =   392.017  mm,	Y =    -5.147  mm,	Z =  2416.121  mm,
	W =     -.021 deg,	P =   -39.773 deg,	R =      .020 deg
   GP2:
	UF : 0, UT : 1,
	J1=    90.000 deg,	J2=   180.000 deg
};
P[1033]{
   GP1:
	UF : 1, UT : 1,
	J1=      .005 deg,	J2=   -44.424 deg,	J3=    65.270 deg,
	J4=      .005 deg,	J5=   -70.270 deg,	J6=     -.002 deg
   GP2:
	UF : 0, UT : 1,
	J1=    90.000 deg,	J2=     0.000 deg
};
P[1034]{
   GP1:
	UF : 1, UT : 1,		CONFIG : 'N U T, 0, 0, 0',
	X =  1819.034  mm,	Y =    -6.897  mm,	Z =   564.314  mm,
	W =     -.000 deg,	P =    45.917 deg,	R =    -2.669 deg
   GP2:
	UF : 0, UT : 1,
	J1=    90.000 deg,	J2=     0.000 deg
};
P[1035]{
   GP1:
	UF : 1, UT : 1,		CONFIG : 'N U T, 0, 0, 0',
	X =  1621.906  mm,	Y =   155.031  mm,	Z =   510.314  mm,
	W =      .000 deg,	P =    45.917 deg,	R =    -2.669 deg
   GP2:
	UF : 0, UT : 1,
	J1=    90.000 deg,	J2=     0.000 deg
};
P[1036]{
   GP1:
	UF : 1, UT : 1,		CONFIG : 'N U T, 0, 0, 0',
	X =  1616.404  mm,	Y =   131.606  mm,	Z =   408.971  mm,
	W =      .067 deg,	P =    45.900 deg,	R =    17.155 deg
   GP2:
	UF : 0, UT : 1,
	J1=    90.000 deg,	J2=      .000 deg
};
P[1037]{
   GP1:
	UF : 1, UT : 1,		CONFIG : 'N U T, 0, 0, 0',
	X =  1617.114  mm,	Y =   141.899  mm,	Z =   409.681  mm,
	W =      .000 deg,	P =    45.917 deg,	R =    -2.669 deg
   GP2:
	UF : 0, UT : 1,
	J1=    90.000 deg,	J2=     0.000 deg
};
P[1038]{
   GP1:
	UF : 1, UT : 1,		CONFIG : 'N U T, 0, 0, 0',
	X =  1617.563  mm,	Y =   221.810  mm,	Z =   410.818  mm,
	W =      .000 deg,	P =    45.918 deg,	R =    -8.452 deg
   GP2:
	UF : 0, UT : 1,
	J1=    90.000 deg,	J2=     0.000 deg
};
P[1039]{
   GP1:
	UF : 1, UT : 1,		CONFIG : 'N U T, 0, 0, 0',
	X =  1653.539  mm,	Y =   314.670  mm,	Z =   458.639  mm,
	W =     -.000 deg,	P =    45.917 deg,	R =    -2.669 deg
   GP2:
	UF : 0, UT : 1,
	J1=    90.000 deg,	J2=     0.000 deg
};
P[1040]{
   GP1:
	UF : 1, UT : 1,		CONFIG : 'N U T, 0, 0, 0',
	X =  1616.796  mm,	Y =   350.032  mm,	Z =   411.226  mm,
	W =     3.791 deg,	P =    48.896 deg,	R =    -1.442 deg
   GP2:
	UF : 0, UT : 1,
	J1=    90.000 deg,	J2=      .000 deg
};
P[1041]{
   GP1:
	UF : 1, UT : 1,		CONFIG : 'N U T, 0, 0, 0',
	X =  1615.694  mm,	Y =   432.338  mm,	Z =   411.156  mm,
	W =    21.553 deg,	P =    45.140 deg,	R =    22.664 deg
   GP2:
	UF : 0, UT : 1,
	J1=    90.000 deg,	J2=     0.000 deg
};
P[1042]{
   GP1:
	UF : 1, UT : 1,		CONFIG : 'N U T, 0, 0, 0',
	X =  1707.541  mm,	Y =   314.671  mm,	Z =   548.639  mm,
	W =    14.296 deg,	P =    44.115 deg,	R =    18.950 deg
   GP2:
	UF : 0, UT : 1,
	J1=    90.000 deg,	J2=     0.000 deg
};
P[1043]{
   GP1:
	UF : 1, UT : 1,		CONFIG : 'N U T, 0, 0, 0',
	X =  1707.539  mm,	Y =  -139.330  mm,	Z =   548.639  mm,
	W =     -.000 deg,	P =    45.919 deg,	R =    -2.669 deg
   GP2:
	UF : 0, UT : 1,
	J1=    90.000 deg,	J2=     0.000 deg
};
P[1044]{
   GP1:
	UF : 1, UT : 1,		CONFIG : 'N U T, 0, 0, 0',
	X =  1614.726  mm,	Y =  -127.279  mm,	Z =   409.297  mm,
	W =      .096 deg,	P =    45.916 deg,	R =    -3.643 deg
   GP2:
	UF : 0, UT : 1,
	J1=    90.000 deg,	J2=      .000 deg
};
P[1045]{
   GP1:
	UF : 1, UT : 1,		CONFIG : 'N U T, 0, 0, 0',
	X =  1614.702  mm,	Y =  -160.882  mm,	Z =   410.034  mm,
	W =      .096 deg,	P =    46.938 deg,	R =     3.751 deg
   GP2:
	UF : 0, UT : 1,
	J1=    90.000 deg,	J2=     0.000 deg
};
P[1046]{
   GP1:
	UF : 1, UT : 1,		CONFIG : 'N U T, 0, 0, 0',
	X =  1613.017  mm,	Y =  -196.806  mm,	Z =   411.621  mm,
	W =     1.031 deg,	P =    48.639 deg,	R =    42.126 deg
   GP2:
	UF : 0, UT : 1,
	J1=    90.000 deg,	J2=     0.000 deg
};
P[1047]{
   GP1:
	UF : 1, UT : 1,		CONFIG : 'N U T, 0, 0, 0',
	X =  1664.805  mm,	Y =  -152.179  mm,	Z =   471.791  mm,
	W =     1.031 deg,	P =    48.639 deg,	R =    42.126 deg
   GP2:
	UF : 0, UT : 1,
	J1=    90.000 deg,	J2=     0.000 deg
};
P[1048]{
   GP1:
	UF : 1, UT : 1,		CONFIG : 'N U T, 0, 0, 0',
	X =  1710.650  mm,	Y =  -235.344  mm,	Z =   518.121  mm,
	W =     -.000 deg,	P =    45.919 deg,	R =    -2.669 deg
   GP2:
	UF : 0, UT : 1,
	J1=    90.000 deg,	J2=     0.000 deg
};
P[1049]{
   GP1:
	UF : 1, UT : 1,		CONFIG : 'N U T, 0, 0, 0',
	X =  1615.648  mm,	Y =  -221.012  mm,	Z =   411.430  mm,
	W =     1.085 deg,	P =    45.398 deg,	R =    -1.563 deg
   GP2:
	UF : 0, UT : 1,
	J1=    90.000 deg,	J2=     0.000 deg
};
P[1050]{
   GP1:
	UF : 1, UT : 1,		CONFIG : 'N U T, 0, 0, 0',
	X =  1615.484  mm,	Y =  -193.298  mm,	Z =   410.211  mm,
	W =     1.093 deg,	P =    45.391 deg,	R =   -28.069 deg
   GP2:
	UF : 0, UT : 1,
	J1=    90.000 deg,	J2=      .000 deg
};
P[1051]{
   GP1:
	UF : 1, UT : 1,		CONFIG : 'N U T, 0, 0, 0',
	X =  1665.750  mm,	Y =  -216.620  mm,	Z =   476.833  mm,
	W =     1.098 deg,	P =    45.401 deg,	R =   -28.069 deg
   GP2:
	UF : 0, UT : 1,
	J1=    89.999 deg,	J2=     0.000 deg
};
P[1052]{
   GP1:
	UF : 1, UT : 1,		CONFIG : 'N U T, 0, 0, 0',
	X =  1710.649  mm,	Y =  -235.344  mm,	Z =   518.121  mm,
	W =     -.000 deg,	P =    45.919 deg,	R =    -2.669 deg
   GP2:
	UF : 0, UT : 1,
	J1=    90.000 deg,	J2=     0.000 deg
};
P[1053]{
   GP1:
	UF : 1, UT : 1,		CONFIG : 'N U T, 0, 0, 0',
	X =  1710.649  mm,	Y =  -335.344  mm,	Z =   518.121  mm,
	W =   -24.937 deg,	P =    39.897 deg,	R =   -38.608 deg
   GP2:
	UF : 0, UT : 1,
	J1=    90.000 deg,	J2=     0.000 deg
};
P[1054]{
   GP1:
	UF : 1, UT : 1,		CONFIG : 'N U T, 0, 0, 0',
	X =  1615.018  mm,	Y =  -353.317  mm,	Z =   411.647  mm,
	W =   -28.551 deg,	P =    41.609 deg,	R =   -35.630 deg
   GP2:
	UF : 0, UT : 1,
	J1=    89.999 deg,	J2=      .000 deg
};
P[1055]{
   GP1:
	UF : 1, UT : 1,		CONFIG : 'N U T, 0, 0, 0',
	X =  1615.298  mm,	Y =  -433.271  mm,	Z =   410.910  mm,
	W =   -28.808 deg,	P =    41.508 deg,	R =   -35.729 deg
   GP2:
	UF : 0, UT : 1,
	J1=    90.000 deg,	J2=     0.000 deg
};
P[1056]{
   GP1:
	UF : 1, UT : 1,		CONFIG : 'N U T, 0, 0, 0',
	X =  1730.632  mm,	Y =  -410.643  mm,	Z =   540.658  mm,
	W =   -30.592 deg,	P =    36.083 deg,	R =   -32.808 deg
   GP2:
	UF : 0, UT : 1,
	J1=    90.000 deg,	J2=     0.000 deg
};
P[1057]{
   GP1:
	UF : 1, UT : 1,		CONFIG : 'N U T, 0, 0, 0',
	X =  1816.930  mm,	Y =  -158.897  mm,	Z =   555.408  mm,
	W =   -13.122 deg,	P =    44.168 deg,	R =   -15.536 deg
   GP2:
	UF : 0, UT : 1,
	J1=    90.000 deg,	J2=     0.000 deg
};
P[1058]{
   GP1:
	UF : 1, UT : 1,		CONFIG : 'N U T, 0, 0, 0',
	X =  1665.514  mm,	Y =   -76.222  mm,	Z =   459.026  mm,
	W =    -1.398 deg,	P =    45.211 deg,	R =    -2.659 deg
   GP2:
	UF : 0, UT : 1,
	J1=    90.000 deg,	J2=     0.000 deg
};
P[1059]{
   GP1:
	UF : 1, UT : 1,		CONFIG : 'N U T, 0, 0, 0',
	X =  1634.638  mm,	Y =   -80.822  mm,	Z =   408.400  mm,
	W =    -1.410 deg,	P =    46.984 deg,	R =     8.231 deg
   GP2:
	UF : 0, UT : 1,
	J1=    90.000 deg,	J2=      .000 deg
};
P[1060]{
   GP1:
	UF : 1, UT : 1,		CONFIG : 'N U T, 0, 0, 0',
	X =  1636.173  mm,	Y =   -49.516  mm,	Z =   408.646  mm,
	W =    -2.439 deg,	P =    46.947 deg,	R =   -13.024 deg
   GP2:
	UF : 0, UT : 1,
	J1=    90.000 deg,	J2=     0.000 deg
};
P[1061]{
   GP1:
	UF : 1, UT : 1,		CONFIG : 'N U T, 0, 0, 0',
	X =  1709.034  mm,	Y =   -60.897  mm,	Z =   538.606  mm,
	W =     -.000 deg,	P =    45.917 deg,	R =    -2.669 deg
   GP2:
	UF : 0, UT : 1,
	J1=    90.000 deg,	J2=     0.000 deg
};
P[1062]{
   GP1:
	UF : 1, UT : 1,		CONFIG : 'N U T, 0, 0, 0',
	X =  1709.034  mm,	Y =    70.103  mm,	Z =   538.605  mm,
	W =     -.000 deg,	P =    45.917 deg,	R =    -2.669 deg
   GP2:
	UF : 0, UT : 1,
	J1=    90.000 deg,	J2=     0.000 deg
};
P[1063]{
   GP1:
	UF : 1, UT : 1,		CONFIG : 'N U T, 0, 0, 0',
	X =  1637.812  mm,	Y =    78.782  mm,	Z =   409.850  mm,
	W =    -1.870 deg,	P =    44.966 deg,	R =    -2.659 deg
   GP2:
	UF : 0, UT : 1,
	J1=    90.000 deg,	J2=     0.000 deg
};
P[1064]{
   GP1:
	UF : 1, UT : 1,		CONFIG : 'N U T, 0, 0, 0',
	X =  1638.070  mm,	Y =    -5.469  mm,	Z =   410.295  mm,
	W =    -1.870 deg,	P =    44.966 deg,	R =    -2.659 deg
   GP2:
	UF : 0, UT : 1,
	J1=    90.000 deg,	J2=     0.000 deg
};
P[1065]{
   GP1:
	UF : 1, UT : 1,		CONFIG : 'N U T, 0, 0, 0',
	X =  1709.034  mm,	Y =    70.103  mm,	Z =   538.605  mm,
	W =     -.000 deg,	P =    45.917 deg,	R =    -2.669 deg
   GP2:
	UF : 0, UT : 1,
	J1=    90.000 deg,	J2=     0.000 deg
};
P[1066]{
   GP1:
	UF : 1, UT : 1,		CONFIG : 'N U T, 0, 0, 0',
	X =  1617.914  mm,	Y =    80.097  mm,	Z =   419.790  mm,
	W =      .021 deg,	P =    45.919 deg,	R =    -2.645 deg
   GP2:
	UF : 0, UT : 1,
	J1=    90.000 deg,	J2=      .000 deg
};
P[1067]{
   GP1:
	UF : 1, UT : 1,		CONFIG : 'N U T, 0, 0, 0',
	X =  1618.329  mm,	Y =    53.421  mm,	Z =   420.061  mm,
	W =    -2.071 deg,	P =    48.970 deg,	R =     -.692 deg
   GP2:
	UF : 0, UT : 1,
	J1=    90.000 deg,	J2=     0.000 deg
};
P[1068]{
   GP1:
	UF : 1, UT : 1,		CONFIG : 'N U T, 0, 0, 0',
	X =  1709.034  mm,	Y =    70.103  mm,	Z =   538.605  mm,
	W =     -.000 deg,	P =    45.917 deg,	R =    -2.669 deg
   GP2:
	UF : 0, UT : 1,
	J1=    90.000 deg,	J2=     0.000 deg
};
P[1069]{
   GP1:
	UF : 1, UT : 1,		CONFIG : 'N U T, 0, 0, 0',
	X =  1709.034  mm,	Y =   -77.897  mm,	Z =   538.605  mm,
	W =     -.000 deg,	P =    45.917 deg,	R =    -2.669 deg
   GP2:
	UF : 0, UT : 1,
	J1=    90.000 deg,	J2=     0.000 deg
};
P[1070]{
   GP1:
	UF : 1, UT : 1,		CONFIG : 'N U T, 0, 0, 0',
	X =  1615.604  mm,	Y =   -81.949  mm,	Z =   419.038  mm,
	W =    -2.076 deg,	P =    48.967 deg,	R =     4.167 deg
   GP2:
	UF : 0, UT : 1,
	J1=    90.000 deg,	J2=     0.000 deg
};
P[1071]{
   GP1:
	UF : 1, UT : 1,		CONFIG : 'N U T, 0, 0, 0',
	X =  1618.037  mm,	Y =   -54.983  mm,	Z =   421.205  mm,
	W =    -2.076 deg,	P =    48.967 deg,	R =    -8.307 deg
   GP2:
	UF : 0, UT : 1,
	J1=    90.000 deg,	J2=     0.000 deg
};
P[1072]{
   GP1:
	UF : 1, UT : 1,		CONFIG : 'N U T, 0, 0, 0',
	X =  1721.744  mm,	Y =   -51.899  mm,	Z =   520.175  mm,
	W =    -2.076 deg,	P =    48.967 deg,	R =    -2.751 deg
   GP2:
	UF : 0, UT : 1,
	J1=    90.000 deg,	J2=     0.000 deg
};
P[1073]{
   GP1:
	UF : 1, UT : 1,		CONFIG : 'N U T, 0, 0, 0',
	X =  1618.744  mm,	Y =    -9.232  mm,	Z =   520.175  mm,
	W =    -2.076 deg,	P =    48.967 deg,	R =    79.079 deg
   GP2:
	UF : 0, UT : 1,
	J1=    90.000 deg,	J2=     0.000 deg
};
P[1074]{
   GP1:
	UF : 1, UT : 1,		CONFIG : 'N U T, 0, 0, 0',
	X =  1611.108  mm,	Y =   -51.241  mm,	Z =   417.692  mm,
	W =    -7.325 deg,	P =    44.527 deg,	R =    79.612 deg
   GP2:
	UF : 0, UT : 1,
	J1=    90.000 deg,	J2=     0.000 deg
};
P[1075]{
   GP1:
	UF : 1, UT : 1,		CONFIG : 'N U T, 0, 0, 0',
	X =  1596.840  mm,	Y =   -51.126  mm,	Z =   417.213  mm,
	W =    -7.325 deg,	P =    44.527 deg,	R =    79.612 deg
   GP2:
	UF : 0, UT : 1,
	J1=    90.000 deg,	J2=     0.000 deg
};
P[1076]{
   GP1:
	UF : 1, UT : 1,		CONFIG : 'N U T, 0, 0, 0',
	X =  1618.744  mm,	Y =    -9.232  mm,	Z =   520.175  mm,
	W =    -2.076 deg,	P =    48.967 deg,	R =    79.079 deg
   GP2:
	UF : 0, UT : 1,
	J1=    90.000 deg,	J2=     0.000 deg
};
P[1077]{
   GP1:
	UF : 1, UT : 1,		CONFIG : 'N U T, 0, 0, 0',
	X =  1618.744  mm,	Y =    26.526  mm,	Z =   520.175  mm,
	W =    -2.076 deg,	P =    48.967 deg,	R =   -94.932 deg
   GP2:
	UF : 0, UT : 1,
	J1=    90.000 deg,	J2=     0.000 deg
};
P[1078]{
   GP1:
	UF : 1, UT : 1,		CONFIG : 'N U T, 0, 0, 0',
	X =  1613.714  mm,	Y =    48.029  mm,	Z =   417.969  mm,
	W =    -3.289 deg,	P =    44.906 deg,	R =   -94.653 deg
   GP2:
	UF : 0, UT : 1,
	J1=    90.000 deg,	J2=     0.000 deg
};
P[1079]{
   GP1:
	UF : 1, UT : 1,		CONFIG : 'N U T, 0, 0, 0',
	X =  1602.075  mm,	Y =    47.944  mm,	Z =   418.495  mm,
	W =    -3.289 deg,	P =    44.905 deg,	R =   -94.653 deg
   GP2:
	UF : 0, UT : 1,
	J1=    90.000 deg,	J2=     0.000 deg
};
P[1080]{
   GP1:
	UF : 1, UT : 1,		CONFIG : 'N U T, 0, 0, 0',
	X =  1618.744  mm,	Y =    26.526  mm,	Z =   520.175  mm,
	W =     -.707 deg,	P =    36.028 deg,	R =   -94.002 deg
   GP2:
	UF : 0, UT : 1,
	J1=    90.000 deg,	J2=     0.000 deg
};
P[1081]{
   GP1:
	UF : 1, UT : 1,		CONFIG : 'N U T, 0, 0, 0',
	X =  2051.968  mm,	Y =  -337.038  mm,	Z =   536.737  mm,
	W =   -45.319 deg,	P =     7.608 deg,	R =     5.072 deg
   GP2:
	UF : 0, UT : 1,
	J1=    90.000 deg,	J2=     0.000 deg
};
P[1082]{
   GP1:
	UF : 1, UT : 1,		CONFIG : 'N U T, 0, 0, 0',
	X =  2065.258  mm,	Y =  -440.562  mm,	Z =   416.925  mm,
	W =   -44.803 deg,	P =     3.316 deg,	R =     4.925 deg
   GP2:
	UF : 1, UT : 1,
	J1=    90.000 deg,	J2=      .000 deg
};
P[1083]{
   GP1:
	UF : 1, UT : 1,		CONFIG : 'N U T, 0, 0, 0',
	X =  2119.404  mm,	Y =  -440.015  mm,	Z =   419.473  mm,
	W =   -44.800 deg,	P =     3.306 deg,	R =     4.922 deg
   GP2:
	UF : 1, UT : 1,
	J1=    90.000 deg,	J2=     0.000 deg
};
P[1084]{
   GP1:
	UF : 1, UT : 1,		CONFIG : 'N U T, 0, 0, 0',
	X =  2165.659  mm,	Y =  -440.071  mm,	Z =   420.450  mm,
	W =   -35.985 deg,	P =     2.077 deg,	R =     4.572 deg
   GP2:
	UF : 1, UT : 1,
	J1=    90.000 deg,	J2=     0.000 deg
};
P[1085]{
   GP1:
	UF : 1, UT : 1,		CONFIG : 'N U T, 0, 0, 0',
	X =  2192.152  mm,	Y =  -439.912  mm,	Z =   420.613  mm,
	W =   -46.529 deg,	P =     3.253 deg,	R =     4.441 deg
   GP2:
	UF : 1, UT : 1,
	J1=    90.000 deg,	J2=     0.000 deg
};
P[1086]{
   GP1:
	UF : 1, UT : 1,		CONFIG : 'N U T, 0, 0, 0',
	X =  2312.005  mm,	Y =  -442.540  mm,	Z =   421.471  mm,
	W =   -44.812 deg,	P =     3.500 deg,	R =     4.729 deg
   GP2:
	UF : 1, UT : 1,
	J1=    90.000 deg,	J2=     0.000 deg
};
P[1087]{
   GP1:
	UF : 1, UT : 1,		CONFIG : 'N U T, 0, 0, 0',
	X =  2322.380  mm,	Y =  -374.657  mm,	Z =   488.435  mm,
	W =   -45.801 deg,	P =     3.717 deg,	R =     4.521 deg
   GP2:
	UF : 0, UT : 1,
	J1=    90.000 deg,	J2=     0.000 deg
};
P[1088]{
   GP1:
	UF : 1, UT : 1,		CONFIG : 'N U T, 0, 0, 0',
	X =  2313.720  mm,	Y =  -422.562  mm,	Z =   410.868  mm,
	W =   -38.970 deg,	P =     1.358 deg,	R =    -8.449 deg
   GP2:
	UF : 1, UT : 1,
	J1=    90.000 deg,	J2=      .000 deg
};
P[1089]{
   GP1:
	UF : 1, UT : 1,		CONFIG : 'N U T, 0, 0, 0',
	X =  2245.266  mm,	Y =  -408.951  mm,	Z =   407.695  mm,
	W =   -42.398 deg,	P =     3.388 deg,	R =   -10.193 deg
   GP2:
	UF : 1, UT : 1,
	J1=    90.000 deg,	J2=      .000 deg
};
P[1090]{
   GP1:
	UF : 1, UT : 1,		CONFIG : 'N U T, 0, 0, 0',
	X =  2157.750  mm,	Y =  -383.025  mm,	Z =   409.230  mm,
	W =   -44.997 deg,	P =      .478 deg,	R =   -16.008 deg
   GP2:
	UF : 1, UT : 1,
	J1=    90.000 deg,	J2=     0.000 deg
};
P[1091]{
   GP1:
	UF : 1, UT : 1,		CONFIG : 'N U T, 0, 0, 0',
	X =  2192.646  mm,	Y =  -316.002  mm,	Z =   488.370  mm,
	W =   -45.800 deg,	P =     3.717 deg,	R =   -19.293 deg
   GP2:
	UF : 0, UT : 1,
	J1=    90.000 deg,	J2=     0.000 deg
};
P[1092]{
   GP1:
	UF : 1, UT : 1,		CONFIG : 'N U T, 0, 0, 0',
	X =  2355.557  mm,	Y =  -374.570  mm,	Z =   640.258  mm,
	W =   -45.370 deg,	P =     3.743 deg,	R =     3.813 deg
   GP2:
	UF : 0, UT : 1,
	J1=    90.000 deg,	J2=     0.000 deg
};
P[1093]{
   GP1:
	UF : 1, UT : 1,		CONFIG : 'N U T, 0, 0, 0',
	X =  2345.996  mm,	Y =  -443.552  mm,	Z =   567.564  mm,
	W =   -44.875 deg,	P =     3.774 deg,	R =     3.782 deg
   GP2:
	UF : 0, UT : 1,
	J1=    90.000 deg,	J2=     0.000 deg
};
P[1094]{
   GP1:
	UF : 1, UT : 1,		CONFIG : 'N U T, 0, 0, 0',
	X =  2398.567  mm,	Y =  -440.723  mm,	Z =   569.133  mm,
	W =   -43.832 deg,	P =    11.293 deg,	R =    25.930 deg
   GP2:
	UF : 0, UT : 1,
	J1=    90.000 deg,	J2=     0.000 deg
};
P[1095]{
   GP1:
	UF : 1, UT : 1,		CONFIG : 'N U T, 0, 0, 0',
	X =  2361.646  mm,	Y =  -316.002  mm,	Z =   705.371  mm,
	W =   -45.800 deg,	P =     3.717 deg,	R =     3.840 deg
   GP2:
	UF : 0, UT : 1,
	J1=    90.000 deg,	J2=     0.000 deg
};
P[1096]{
   GP1:
	UF : 1, UT : 1,		CONFIG : 'N U T, 0, 0, 0',
	X =  2431.558  mm,	Y =  -405.370  mm,	Z =   705.370  mm,
	W =   -45.800 deg,	P =     3.717 deg,	R =     3.840 deg
   GP2:
	UF : 0, UT : 1,
	J1=    90.000 deg,	J2=     0.000 deg
};
P[1097]{
   GP1:
	UF : 1, UT : 1,		CONFIG : 'N U T, 0, 0, 0',
	X =  2479.192  mm,	Y =  -441.664  mm,	Z =   619.931  mm,
	W =   -44.875 deg,	P =     3.774 deg,	R =     3.782 deg
   GP2:
	UF : 0, UT : 1,
	J1=    90.000 deg,	J2=     0.000 deg
};
P[1098]{
   GP1:
	UF : 1, UT : 1,		CONFIG : 'N U T, 0, 0, 0',
	X =  2431.611  mm,	Y =  -442.129  mm,	Z =   618.230  mm,
	W =   -44.875 deg,	P =     3.774 deg,	R =     3.782 deg
   GP2:
	UF : 0, UT : 1,
	J1=    90.000 deg,	J2=     0.000 deg
};
P[1099]{
   GP1:
	UF : 1, UT : 1,		CONFIG : 'N U T, 0, 0, 0',
	X =  2422.708  mm,	Y =  -443.303  mm,	Z =   616.150  mm,
	W =   -47.202 deg,	P =    -4.228 deg,	R =    12.058 deg
   GP2:
	UF : 0, UT : 1,
	J1=    90.000 deg,	J2=     0.000 deg
};
P[1100]{
   GP1:
	UF : 1, UT : 1,		CONFIG : 'N U T, 0, 0, 0',
	X =  2414.079  mm,	Y =  -439.978  mm,	Z =   614.077  mm,
	W =   -54.121 deg,	P =   -12.107 deg,	R =    21.739 deg
   GP2:
	UF : 0, UT : 1,
	J1=    90.000 deg,	J2=     0.000 deg
};
P[1101]{
   GP1:
	UF : 1, UT : 1,		CONFIG : 'N U T, 0, 0, 0',
	X =  2482.296  mm,	Y =  -242.980  mm,	Z =   687.983  mm,
	W =   -45.800 deg,	P =     3.717 deg,	R =     3.840 deg
   GP2:
	UF : 0, UT : 1,
	J1=    90.000 deg,	J2=     0.000 deg
};
P[1102]{
   GP1:
	UF : 1, UT : 1,		CONFIG : 'N U T, 0, 0, 0',
	X =  2505.422  mm,	Y =  -353.441  mm,	Z =   558.985  mm,
	W =   -28.620 deg,	P =   -37.578 deg,	R =   -47.947 deg
   GP2:
	UF : 0, UT : 1,
	J1=    90.000 deg,	J2=     0.000 deg
};
P[1103]{
   GP1:
	UF : 1, UT : 1,		CONFIG : 'N U T, 0, 0, 0',
	X =  2479.805  mm,	Y =  -440.598  mm,	Z =   518.552  mm,
	W =     -.765 deg,	P =   -44.982 deg,	R =   -88.916 deg
   GP2:
	UF : 0, UT : 1,
	J1=    90.000 deg,	J2=      .000 deg
};
P[1104]{
   GP1:
	UF : 1, UT : 1,		CONFIG : 'N U T, 0, 0, 0',
	X =  2431.875  mm,	Y =  -440.714  mm,	Z =   516.919  mm,
	W =   -46.020 deg,	P =   -32.709 deg,	R =   -60.051 deg
   GP2:
	UF : 0, UT : 1,
	J1=    90.000 deg,	J2=     0.000 deg
};
P[1105]{
   GP1:
	UF : 1, UT : 1,		CONFIG : 'N U T, 0, 0, 0',
	X =  2567.563  mm,	Y =  -374.906  mm,	Z =   592.469  mm,
	W =   -28.619 deg,	P =   -37.577 deg,	R =   -73.349 deg
   GP2:
	UF : 0, UT : 1,
	J1=    90.000 deg,	J2=     0.000 deg
};
P[1106]{
   GP1:
	UF : 1, UT : 1,		CONFIG : 'N U T, 0, 0, 0',
	X =  2567.563  mm,	Y =  -194.906  mm,	Z =   592.469  mm,
	W =   -28.619 deg,	P =   -37.577 deg,	R =   -18.464 deg
   GP2:
	UF : 0, UT : 1,
	J1=    90.000 deg,	J2=     0.000 deg
};
P[1107]{
   GP1:
	UF : 1, UT : 1,		CONFIG : 'N U T, 0, 0, 0',
	X =  2072.645  mm,	Y =   372.998  mm,	Z =   516.371  mm,
	W =    43.428 deg,	P =    16.677 deg,	R =   -20.967 deg
   GP2:
	UF : 0, UT : 1,
	J1=    90.000 deg,	J2=     0.000 deg
};
P[1108]{
   GP1:
	UF : 1, UT : 1,		CONFIG : 'N U T, 0, 0, 0',
	X =  2067.494  mm,	Y =   433.863  mm,	Z =   417.870  mm,
	W =    43.968 deg,	P =    11.983 deg,	R =   -17.454 deg
   GP2:
	UF : 1, UT : 1,
	J1=    90.000 deg,	J2=     0.000 deg
};
P[1109]{
   GP1:
	UF : 1, UT : 1,		CONFIG : 'N U T, 0, 0, 0',
	X =  2311.792  mm,	Y =   436.788  mm,	Z =   418.985  mm,
	W =    44.829 deg,	P =     9.277 deg,	R =   -17.295 deg
   GP2:
	UF : 1, UT : 1,
	J1=    90.000 deg,	J2=     0.000 deg
};
P[1110]{
   GP1:
	UF : 1, UT : 1,		CONFIG : 'N U T, 0, 0, 0',
	X =  2310.163  mm,	Y =   364.504  mm,	Z =   487.755  mm,
	W =    43.428 deg,	P =    16.677 deg,	R =   -18.246 deg
   GP2:
	UF : 0, UT : 1,
	J1=    90.000 deg,	J2=     0.000 deg
};
P[1111]{
   GP1:
	UF : 1, UT : 1,		CONFIG : 'N U T, 0, 0, 0',
	X =  2311.278  mm,	Y =   412.063  mm,	Z =   410.676  mm,
	W =    36.139 deg,	P =    15.180 deg,	R =    -9.294 deg
   GP2:
	UF : 1, UT : 1,
	J1=    90.000 deg,	J2=     0.000 deg
};
P[1112]{
   GP1:
	UF : 1, UT : 1,		CONFIG : 'N U T, 0, 0, 0',
	X =  2238.371  mm,	Y =   398.622  mm,	Z =   408.876  mm,
	W =    35.632 deg,	P =    15.709 deg,	R =    -5.398 deg
   GP2:
	UF : 1, UT : 1,
	J1=    90.000 deg,	J2=     0.000 deg
};
P[1113]{
   GP1:
	UF : 1, UT : 1,		CONFIG : 'N U T, 0, 0, 0',
	X =  2157.868  mm,	Y =   378.363  mm,	Z =   408.912  mm,
	W =    42.416 deg,	P =    16.706 deg,	R =     -.979 deg
   GP2:
	UF : 1, UT : 1,
	J1=    90.000 deg,	J2=     0.000 deg
};
P[1114]{
   GP1:
	UF : 1, UT : 1,		CONFIG : 'N U T, 0, 0, 0',
	X =  2183.068  mm,	Y =   301.712  mm,	Z =   672.802  mm,
	W =    43.428 deg,	P =    16.677 deg,	R =    -1.009 deg
   GP2:
	UF : 0, UT : 1,
	J1=    90.000 deg,	J2=     0.000 deg
};
P[1115]{
   GP1:
	UF : 1, UT : 1,		CONFIG : 'N U T, 0, 0, 0',
	X =  2360.068  mm,	Y =   359.712  mm,	Z =   672.802  mm,
	W =    43.428 deg,	P =    16.677 deg,	R =   -16.431 deg
   GP2:
	UF : 0, UT : 1,
	J1=    90.000 deg,	J2=     0.000 deg
};
P[1116]{
   GP1:
	UF : 1, UT : 1,		CONFIG : 'N U T, 0, 0, 0',
	X =  2345.842  mm,	Y =   435.904  mm,	Z =   568.233  mm,
	W =    41.490 deg,	P =    15.419 deg,	R =   -19.151 deg
   GP2:
	UF : 0, UT : 1,
	J1=    90.000 deg,	J2=     0.000 deg
};
P[1117]{
   GP1:
	UF : 1, UT : 1,		CONFIG : 'N U T, 0, 0, 0',
	X =  2400.895  mm,	Y =   434.403  mm,	Z =   569.877  mm,
	W =    40.052 deg,	P =    21.818 deg,	R =   -37.758 deg
   GP2:
	UF : 0, UT : 1,
	J1=    89.994 deg,	J2=      .000 deg
};
P[1118]{
   GP1:
	UF : 1, UT : 1,		CONFIG : 'N U T, 0, 0, 0',
	X =  2360.068  mm,	Y =   359.712  mm,	Z =   672.802  mm,
	W =    43.428 deg,	P =    16.677 deg,	R =   -18.155 deg
   GP2:
	UF : 0, UT : 1,
	J1=    90.000 deg,	J2=     0.000 deg
};
P[1119]{
   GP1:
	UF : 1, UT : 1,		CONFIG : 'N U T, 0, 0, 0',
	X =  2481.175  mm,	Y =   436.218  mm,	Z =   621.065  mm,
	W =    42.312 deg,	P =    17.019 deg,	R =   -17.824 deg
   GP2:
	UF : 0, UT : 1,
	J1=    90.000 deg,	J2=     0.000 deg
};
P[1120]{
   GP1:
	UF : 1, UT : 1,		CONFIG : 'N U T, 0, 0, 0',
	X =  2433.042  mm,	Y =   436.690  mm,	Z =   618.993  mm,
	W =    42.312 deg,	P =    17.019 deg,	R =   -17.824 deg
   GP2:
	UF : 0, UT : 1,
	J1=    90.000 deg,	J2=     0.000 deg
};
P[1121]{
   GP1:
	UF : 1, UT : 1,		CONFIG : 'N U T, 0, 0, 0',
	X =  2421.784  mm,	Y =   436.442  mm,	Z =   618.196  mm,
	W =    46.025 deg,	P =     5.793 deg,	R =   -20.933 deg
   GP2:
	UF : 0, UT : 1,
	J1=    90.000 deg,	J2=     0.000 deg
};
P[1122]{
   GP1:
	UF : 1, UT : 1,		CONFIG : 'N U T, 0, 0, 0',
	X =  2414.343  mm,	Y =   434.635  mm,	Z =   615.173  mm,
	W =    55.585 deg,	P =     -.623 deg,	R =   -30.576 deg
   GP2:
	UF : 0, UT : 1,
	J1=    90.000 deg,	J2=     0.000 deg
};
P[1123]{
   GP1:
	UF : 1, UT : 1,		CONFIG : 'N U T, 0, 0, 0',
	X =  2394.816  mm,	Y =   386.818  mm,	Z =   645.562  mm,
	W =    55.585 deg,	P =     -.624 deg,	R =   -30.576 deg
   GP2:
	UF : 0, UT : 1,
	J1=    90.000 deg,	J2=     0.000 deg
};
P[1124]{
   GP1:
	UF : 1, UT : 1,		CONFIG : 'N U T, 0, 0, 0',
	X =  2512.528  mm,	Y =   214.847  mm,	Z =   694.890  mm,
	W =    45.884 deg,	P =    -1.983 deg,	R =      .633 deg
   GP2:
	UF : 0, UT : 1,
	J1=    90.000 deg,	J2=     0.000 deg
};
P[1125]{
   GP1:
	UF : 1, UT : 1,		CONFIG : 'N U T, 0, 0, 0',
	X =  2512.528  mm,	Y =   371.847  mm,	Z =   563.889  mm,
	W =    28.310 deg,	P =   -37.796 deg,	R =    47.397 deg
   GP2:
	UF : 0, UT : 1,
	J1=    90.000 deg,	J2=     0.000 deg
};
P[1126]{
   GP1:
	UF : 1, UT : 1,		CONFIG : 'N U T, 0, 0, 0',
	X =  2475.852  mm,	Y =   435.206  mm,	Z =   520.599  mm,
	W =     4.772 deg,	P =   -44.999 deg,	R =    96.138 deg
   GP2:
	UF : 0, UT : 1,
	J1=    90.000 deg,	J2=     0.000 deg
};
P[1127]{
   GP1:
	UF : 1, UT : 1,		CONFIG : 'N U T, 0, 0, 0',
	X =  2428.390  mm,	Y =   437.121  mm,	Z =   518.474  mm,
	W =    13.020 deg,	P =   -51.322 deg,	R =    91.635 deg
   GP2:
	UF : 0, UT : 1,
	J1=    90.000 deg,	J2=      .000 deg
};
P[1128]{
   GP1:
	UF : 1, UT : 1,		CONFIG : 'N U T, 0, 0, 0',
	X =  2488.844  mm,	Y =   381.884  mm,	Z =   524.273  mm,
	W =    12.001 deg,	P =   -51.332 deg,	R =    88.206 deg
   GP2:
	UF : 0, UT : 1,
	J1=    90.000 deg,	J2=     0.000 deg
};
P[1129]{
   GP1:
	UF : 1, UT : 1,		CONFIG : 'N U T, 0, 0, 0',
	X =  2531.727  mm,	Y =   371.847  mm,	Z =   563.889  mm,
	W =    28.310 deg,	P =   -37.796 deg,	R =    47.397 deg
   GP2:
	UF : 0, UT : 1,
	J1=    90.000 deg,	J2=     0.000 deg
};
P[1130]{
   GP1:
	UF : 1, UT : 1,		CONFIG : 'N U T, 0, 0, 0',
	X =  2512.528  mm,	Y =    40.847  mm,	Z =   705.891  mm,
	W =    43.428 deg,	P =    16.677 deg,	R =   -18.155 deg
   GP2:
	UF : 0, UT : 1,
	J1=    90.000 deg,	J2=     0.000 deg
};
P[1131]{
   GP1:
	UF : 1, UT : 1,		CONFIG : 'N U T, 0, 0, 0',
	X =  1841.526  mm,	Y =    83.901  mm,	Z =   705.890  mm,
	W =    -6.286 deg,	P =    45.581 deg,	R =  -100.055 deg
   GP2:
	UF : 0, UT : 1,
	J1=    90.000 deg,	J2=     0.000 deg
};
P[1132]{
   GP1:
	UF : 1, UT : 1,		CONFIG : 'N U B, 0, 0, 0',
	X =   357.524  mm,	Y =     -.905  mm,	Z =  2424.587  mm,
	W =     -.002 deg,	P =   -40.002 deg,	R =      .017 deg
   GP2:
	UF : 1, UT : 1,
	J1=    90.000 deg,	J2=      .000 deg
};
P[1133]{
   GP1:
	UF : 1, UT : 1,		CONFIG : 'N U T, 0, 0, 0',
	X =   254.446  mm,	Y =   662.476  mm,	Z =  2161.953  mm,
	W =     -.015 deg,	P =   -26.755 deg,	R =    72.877 deg
   GP2:
	UF : 0, UT : 1,
	J1=    90.000 deg,	J2=     0.000 deg
};
P[1134]{
   GP1:
	UF : 1, UT : 1,		CONFIG : 'N U T, 0, 0, 0',
	X =  1172.993  mm,	Y =  1396.463  mm,	Z =  1371.229  mm,
	W =     2.123 deg,	P =   -27.834 deg,	R =    46.073 deg
   GP2:
	UF : 0, UT : 1,
	J1=    90.000 deg,	J2=    90.000 deg
};
P[1135]{
   GP1:
	UF : 1, UT : 1,		CONFIG : 'N U T, 0, 0, 0',
	X =  2163.792  mm,	Y =  1336.078  mm,	Z =   473.472  mm,
	W =     3.095 deg,	P =    -8.630 deg,	R =    30.802 deg
   GP2:
	UF : 0, UT : 1,
	J1=    90.000 deg,	J2=    90.000 deg
};
P[1136]{
   GP1:
	UF : 1, UT : 1,		CONFIG : 'N U T, 0, 0, 0',
	X =  2799.519  mm,	Y =  1395.574  mm,	Z =    33.669  mm,
	W =      .013 deg,	P =      .004 deg,	R =    23.419 deg
   GP2:
	UF : 0, UT : 1,
	J1=    90.000 deg,	J2=    90.000 deg
};
P[1137]{
   GP1:
	UF : 1, UT : 1,		CONFIG : 'N U T, 0, 0, 0',
	X =  2810.415  mm,	Y =  1434.242  mm,	Z =   -20.801  mm,
	W =      .010 deg,	P =      .014 deg,	R =    23.415 deg
   GP2:
	UF : 1, UT : 1,
	J1=    90.000 deg,	J2=    90.000 deg
};
P[1138]{
   GP1:
	UF : 1, UT : 1,		CONFIG : 'N U T, 0, 0, 0',
	X =  2810.415  mm,	Y =  1434.241  mm,	Z =   -20.801  mm,
	W =      .010 deg,	P =      .014 deg,	R =    23.415 deg
   GP2:
	UF : 1, UT : 1,
	J1=    90.000 deg,	J2=    90.000 deg
};
P[1139]{
   GP1:
	UF : 1, UT : 1,		CONFIG : 'N U T, 0, 0, 0',
	X =  2782.021  mm,	Y =  1413.818  mm,	Z =   -22.817  mm,
	W =      .004 deg,	P =      .014 deg,	R =    23.420 deg
   GP2:
	UF : 1, UT : 1,
	J1=    90.000 deg,	J2=    90.000 deg
};
P[1140]{
   GP1:
	UF : 1, UT : 1,		CONFIG : 'N U T, 0, 0, 0',
	X =  2810.307  mm,	Y =  1413.819  mm,	Z =   -25.174  mm,
	W =      .004 deg,	P =      .014 deg,	R =    23.420 deg
   GP2:
	UF : 1, UT : 1,
	J1=    90.000 deg,	J2=    90.000 deg
};
P[1141]{
   GP1:
	UF : 1, UT : 1,		CONFIG : 'N U T, 0, 0, 0',
	X =  2810.266  mm,	Y =  1413.884  mm,	Z =   -25.278  mm,
	W =      .011 deg,	P =      .017 deg,	R =    23.416 deg
   GP2:
	UF : 1, UT : 1,
	J1=    89.999 deg,	J2=    90.000 deg
};
P[1142]{
   GP1:
	UF : 1, UT : 1,		CONFIG : 'N U T, 0, 0, 0',
	X =  2760.411  mm,	Y =  1423.182  mm,	Z =   -21.552  mm,
	W =      .001 deg,	P =      .017 deg,	R =    23.421 deg
   GP2:
	UF : 1, UT : 1,
	J1=    89.999 deg,	J2=    90.000 deg
};
P[1143]{
   GP1:
	UF : 1, UT : 1,		CONFIG : 'N U T, 0, 0, 0',
	X =  2790.524  mm,	Y =  1423.286  mm,	Z =   -25.530  mm,
	W =      .025 deg,	P =      .021 deg,	R =    23.412 deg
   GP2:
	UF : 1, UT : 1,
	J1=    89.999 deg,	J2=    90.000 deg
};
P[1144]{
   GP1:
	UF : 1, UT : 1,		CONFIG : 'N U T, 0, 0, 0',
	X =  2790.486  mm,	Y =  1423.336  mm,	Z =   -25.637  mm,
	W =      .031 deg,	P =      .024 deg,	R =    23.409 deg
   GP2:
	UF : 1, UT : 1,
	J1=    89.999 deg,	J2=    90.000 deg
};
P[1145]{
   GP1:
	UF : 1, UT : 1,		CONFIG : 'N U T, 0, 0, 0',
	X =  2799.574  mm,	Y =  1430.502  mm,	Z =    52.293  mm,
	W =      .000 deg,	P =      .000 deg,	R =    23.425 deg
   GP2:
	UF : 0, UT : 1,
	J1=    90.000 deg,	J2=    90.000 deg
};
P[1146]{
   GP1:
	UF : 1, UT : 1,		CONFIG : 'N U T, 0, 0, 0',
	X =  2554.369  mm,	Y =  1342.105  mm,	Z =   119.187  mm,
	W =    -1.924 deg,	P =     1.808 deg,	R =    25.005 deg
   GP2:
	UF : 0, UT : 1,
	J1=    90.000 deg,	J2=    90.000 deg
};
P[1147]{
   GP1:
	UF : 1, UT : 1,		CONFIG : 'N U T, 0, 0, 0',
	X =  1405.859  mm,	Y =   227.456  mm,	Z =    82.002  mm,
	W =   -43.796 deg,	P =    -2.383 deg,	R =    15.668 deg
   GP2:
	UF : 0, UT : 1,
	J1=    90.000 deg,	J2=    90.000 deg
};
P[1148]{
   GP1:
	UF : 1, UT : 1,
	J1=    12.539 deg,	J2=   -45.970 deg,	J3=   -23.422 deg,
	J4=    72.490 deg,	J5=   -28.075 deg,	J6=   -34.269 deg
   GP2:
	UF : 0, UT : 1,
	J1=    90.000 deg,	J2=    90.000 deg
};
P[1149]{
   GP1:
	UF : 1, UT : 1,
	J1=    10.219 deg,	J2=   -37.730 deg,	J3=   -29.437 deg,
	J4=    82.467 deg,	J5=   -30.708 deg,	J6=   -48.036 deg
   GP2:
	UF : 1, UT : 1,
	J1=    90.000 deg,	J2=    90.000 deg
};
P[1150]{
   GP1:
	UF : 1, UT : 1,		CONFIG : 'N U T, 0, 0, 0',
	X =  1491.964  mm,	Y =   -31.411  mm,	Z =   -43.028  mm,
	W =   -44.735 deg,	P =     5.500 deg,	R =    17.525 deg
   GP2:
	UF : 1, UT : 1,
	J1=    90.000 deg,	J2=    90.000 deg
};
P[1151]{
   GP1:
	UF : 1, UT : 1,		CONFIG : 'N U T, 0, 0, 0',
	X =  1499.626  mm,	Y =   -26.042  mm,	Z =   -37.552  mm,
	W =   -49.947 deg,	P =   -21.098 deg,	R =    25.385 deg
   GP2:
	UF : 1, UT : 1,
	J1=    90.000 deg,	J2=    90.000 deg
};
P[1152]{
   GP1:
	UF : 1, UT : 1,		CONFIG : 'N U T, 1, 0, 0',
	X =  1503.825  mm,	Y =   -13.700  mm,	Z =   -38.379  mm,
	W =   -46.116 deg,	P =   -26.310 deg,	R =    32.911 deg
   GP2:
	UF : 1, UT : 1,
	J1=    90.000 deg,	J2=    90.000 deg
};
P[1153]{
   GP1:
	UF : 1, UT : 1,		CONFIG : 'N U T, 1, 0, 0',
	X =  1508.466  mm,	Y =    26.902  mm,	Z =   -38.356  mm,
	W =   -42.788 deg,	P =   -29.205 deg,	R =    35.275 deg
   GP2:
	UF : 1, UT : 1,
	J1=    89.999 deg,	J2=    90.000 deg
};
P[1154]{
   GP1:
	UF : 1, UT : 1,		CONFIG : 'N U T, 0, 0, 0',
	X =  1522.816  mm,	Y =    49.684  mm,	Z =   -39.779  mm,
	W =   -40.568 deg,	P =   -21.329 deg,	R =    13.837 deg
   GP2:
	UF : 1, UT : 1,
	J1=    89.999 deg,	J2=    90.000 deg
};
P[1155]{
   GP1:
	UF : 1, UT : 1,		CONFIG : 'N U T, 0, 0, 0',
	X =  1549.361  mm,	Y =    43.427  mm,	Z =   -40.544  mm,
	W =   -38.930 deg,	P =   -14.843 deg,	R =   -39.791 deg
   GP2:
	UF : 1, UT : 1,
	J1=    89.998 deg,	J2=    90.000 deg
};
P[1156]{
   GP1:
	UF : 1, UT : 1,		CONFIG : 'N U T, 0, 0, 0',
	X =  1579.623  mm,	Y =    14.358  mm,	Z =   -40.386  mm,
	W =   -38.918 deg,	P =   -14.837 deg,	R =   -39.804 deg
   GP2:
	UF : 1, UT : 1,
	J1=    89.998 deg,	J2=    90.000 deg
};
P[1157]{
   GP1:
	UF : 1, UT : 1,		CONFIG : 'N U T, 0, 0, 0',
	X =  1586.813  mm,	Y =     8.624  mm,	Z =   -39.542  mm,
	W =   -38.918 deg,	P =   -14.837 deg,	R =   -26.710 deg
   GP2:
	UF : 1, UT : 1,
	J1=    89.998 deg,	J2=    90.000 deg
};
P[1158]{
   GP1:
	UF : 1, UT : 1,		CONFIG : 'N U T, 0, 0, 0',
	X =  1595.263  mm,	Y =     9.389  mm,	Z =   -39.982  mm,
	W =   -38.918 deg,	P =   -14.837 deg,	R =   -13.026 deg
   GP2:
	UF : 1, UT : 1,
	J1=    89.998 deg,	J2=    90.000 deg
};
P[1159]{
   GP1:
	UF : 1, UT : 1,		CONFIG : 'N U T, 0, 0, 0',
	X =  1582.254  mm,	Y =   163.348  mm,	Z =     9.339  mm,
	W =   -43.745 deg,	P =    -3.325 deg,	R =    -4.329 deg
   GP2:
	UF : 0, UT : 1,
	J1=    90.000 deg,	J2=    90.000 deg
};
P[1160]{
   GP1:
	UF : 1, UT : 1,		CONFIG : 'N U T, 0, 0, 0',
	X =  1685.374  mm,	Y =   285.724  mm,	Z =    20.813  mm,
	W =    54.391 deg,	P =     4.756 deg,	R =   -78.540 deg
   GP2:
	UF : 0, UT : 1,
	J1=    90.000 deg,	J2=    90.000 deg
};
P[1161]{
   GP1:
	UF : 1, UT : 1,		CONFIG : 'N U T, 0, 0, 0',
	X =  1921.374  mm,	Y =    85.725  mm,	Z =    19.097  mm,
	W =    44.321 deg,	P =     6.701 deg,	R =   -79.548 deg
   GP2:
	UF : 0, UT : 1,
	J1=    90.000 deg,	J2=    90.000 deg
};
P[1162]{
   GP1:
	UF : 1, UT : 1,		CONFIG : 'N U T, 0, 0, 0',
	X =  2023.221  mm,	Y =    46.932  mm,	Z =   -37.754  mm,
	W =    44.242 deg,	P =    16.885 deg,	R =  -113.422 deg
   GP2:
	UF : 0, UT : 1,
	J1=    90.000 deg,	J2=    90.000 deg
};
P[1163]{
   GP1:
	UF : 1, UT : 1,		CONFIG : 'N U T, 0, 0, -1',
	X =  2042.831  mm,	Y =    17.807  mm,	Z =   -36.270  mm,
	W =    48.943 deg,	P =    10.738 deg,	R =  -117.194 deg
   GP2:
	UF : 0, UT : 1,
	J1=    90.000 deg,	J2=    90.000 deg
};
P[1164]{
   GP1:
	UF : 1, UT : 1,		CONFIG : 'N U T, 0, 0, -1',
	X =  1877.442  mm,	Y =    81.577  mm,	Z =    79.657  mm,
	W =    40.231 deg,	P =    21.454 deg,	R =  -138.980 deg
   GP2:
	UF : 0, UT : 1,
	J1=    90.000 deg,	J2=    90.000 deg
};
P[1165]{
   GP1:
	UF : 1, UT : 1,		CONFIG : 'N U T, 0, 0, 0',
	X =   704.218  mm,	Y =   388.449  mm,	Z =   -44.585  mm,
	W =   -14.827 deg,	P =    66.137 deg,	R =     2.515 deg
   GP2:
	UF : 0, UT : 1,
	J1=    90.000 deg,	J2=    90.000 deg
};
P[1166]{
   GP1:
	UF : 1, UT : 1,		CONFIG : 'N U T, 0, 0, 0',
	X =  1237.254  mm,	Y =  -447.653  mm,	Z =     9.338  mm,
	W =    33.676 deg,	P =    29.929 deg,	R =    49.697 deg
   GP2:
	UF : 0, UT : 1,
	J1=    90.000 deg,	J2=    90.000 deg
};
P[1167]{
   GP1:
	UF : 1, UT : 1,		CONFIG : 'N U T, 0, 0, 0',
	X =   879.900  mm,	Y =   -86.392  mm,	Z =   -19.084  mm,
	W =    43.573 deg,	P =    69.244 deg,	R =    28.521 deg
   GP2:
	UF : 0, UT : 1,
	J1=    90.000 deg,	J2=    90.000 deg
};
P[1168]{
   GP1:
	UF : 1, UT : 1,		CONFIG : 'N U T, 0, 0, 0',
	X =  1543.398  mm,	Y =  -219.276  mm,	Z =   139.295  mm,
	W =    51.798 deg,	P =    44.095 deg,	R =    47.739 deg
   GP2:
	UF : 0, UT : 1,
	J1=    90.000 deg,	J2=    90.000 deg
};
P[1169]{
   GP1:
	UF : 1, UT : 1,		CONFIG : 'N U T, 0, 0, 0',
	X =  1706.625  mm,	Y =  -444.344  mm,	Z =     3.766  mm,
	W =    13.040 deg,	P =    46.585 deg,	R =    21.075 deg
   GP2:
	UF : 0, UT : 1,
	J1=    90.000 deg,	J2=    90.000 deg
};
P[1170]{
   GP1:
	UF : 1, UT : 1,		CONFIG : 'N U T, 0, 0, 0',
	X =  1683.570  mm,	Y =  -491.040  mm,	Z =   -42.200  mm,
	W =     5.245 deg,	P =    44.744 deg,	R =    15.369 deg
   GP2:
	UF : 1, UT : 1,
	J1=    90.000 deg,	J2=    90.000 deg
};
P[1171]{
   GP1:
	UF : 1, UT : 1,		CONFIG : 'N U T, 0, 0, 0',
	X =  1619.148  mm,	Y =   -22.429  mm,	Z =   -41.681  mm,
	W =    39.719 deg,	P =    23.175 deg,	R =    65.389 deg
   GP2:
	UF : 1, UT : 1,
	J1=    90.000 deg,	J2=    90.000 deg
};
P[1172]{
   GP1:
	UF : 1, UT : 1,		CONFIG : 'N U T, 0, 0, 0',
	X =  1684.796  mm,	Y =  -168.096  mm,	Z =   107.228  mm,
	W =    41.445 deg,	P =    15.816 deg,	R =    42.913 deg
   GP2:
	UF : 0, UT : 1,
	J1=    90.000 deg,	J2=    90.000 deg
};
P[1173]{
   GP1:
	UF : 1, UT : 1,		CONFIG : 'N U T, 0, 0, -1',
	X =  1926.362  mm,	Y =  -139.788  mm,	Z =   193.210  mm,
	W =   -31.942 deg,	P =   -31.595 deg,	R =    87.860 deg
   GP2:
	UF : 0, UT : 1,
	J1=    75.000 deg,	J2=    90.000 deg
};
P[1174]{
   GP1:
	UF : 1, UT : 1,		CONFIG : 'N U T, 0, 0, -1',
	X =  1953.942  mm,	Y =   -11.283  mm,	Z =    34.184  mm,
	W =   -32.683 deg,	P =    -8.616 deg,	R =   124.477 deg
   GP2:
	UF : 1, UT : 1,
	J1=    75.000 deg,	J2=    90.000 deg
};
P[1175]{
   GP1:
	UF : 1, UT : 1,		CONFIG : 'N U T, 0, 0, -1',
	X =  1992.866  mm,	Y =   -67.843  mm,	Z =    22.749  mm,
	W =   -25.390 deg,	P =   -11.829 deg,	R =   119.523 deg
   GP2:
	UF : 1, UT : 1,
	J1=    75.000 deg,	J2=    90.000 deg
};
P[1176]{
   GP1:
	UF : 1, UT : 1,		CONFIG : 'N U T, 0, 0, -1',
	X =  2021.982  mm,	Y =  -111.483  mm,	Z =    15.539  mm,
	W =   -24.058 deg,	P =   -19.420 deg,	R =   107.017 deg
   GP2:
	UF : 1, UT : 1,
	J1=    75.000 deg,	J2=    90.000 deg
};
P[1177]{
   GP1:
	UF : 1, UT : 1,		CONFIG : 'N U T, 0, 0, -1',
	X =  2031.545  mm,	Y =  -119.748  mm,	Z =    10.887  mm,
	W =   -27.470 deg,	P =   -20.247 deg,	R =   103.965 deg
   GP2:
	UF : 1, UT : 1,
	J1=    75.000 deg,	J2=    90.000 deg
};
P[1178]{
   GP1:
	UF : 1, UT : 1,		CONFIG : 'N U T, 0, 0, -1',
	X =  2038.384  mm,	Y =  -131.652  mm,	Z =    10.692  mm,
	W =   -29.318 deg,	P =   -23.368 deg,	R =   119.590 deg
   GP2:
	UF : 1, UT : 1,
	J1=    75.000 deg,	J2=    90.000 deg
};
P[1179]{
   GP1:
	UF : 1, UT : 1,		CONFIG : 'N U T, 0, 0, -1',
	X =  2054.196  mm,	Y =  -142.577  mm,	Z =     6.271  mm,
	W =   -27.176 deg,	P =   -31.299 deg,	R =   125.406 deg
   GP2:
	UF : 1, UT : 1,
	J1=    75.000 deg,	J2=    90.000 deg
};
P[1180]{
   GP1:
	UF : 1, UT : 1,		CONFIG : 'N U T, 0, 0, -1',
	X =  2138.616  mm,	Y =  -185.620  mm,	Z =   -14.688  mm,
	W =   -28.856 deg,	P =   -29.793 deg,	R =   128.699 deg
   GP2:
	UF : 0, UT : 1,
	J1=    75.000 deg,	J2=    90.000 deg
};
P[1181]{
   GP1:
	UF : 1, UT : 1,		CONFIG : 'N U T, 0, 0, -1',
	X =  2151.849  mm,	Y =  -193.767  mm,	Z =   -18.067  mm,
	W =   -25.181 deg,	P =   -29.053 deg,	R =   112.956 deg
   GP2:
	UF : 0, UT : 1,
	J1=    75.000 deg,	J2=    90.000 deg
};
P[1182]{
   GP1:
	UF : 1, UT : 1,		CONFIG : 'N U T, 0, 0, -1',
	X =  2309.475  mm,	Y =  -313.678  mm,	Z =   -58.656  mm,
	W =   -35.809 deg,	P =   -12.717 deg,	R =   141.916 deg
   GP2:
	UF : 0, UT : 1,
	J1=    75.000 deg,	J2=    90.000 deg
};
P[1183]{
   GP1:
	UF : 1, UT : 1,		CONFIG : 'N U T, 0, 0, -1',
	X =  2332.141  mm,	Y =  -338.485  mm,	Z =   -65.977  mm,
	W =   -32.127 deg,	P =     2.702 deg,	R =   131.528 deg
   GP2:
	UF : 0, UT : 1,
	J1=    75.000 deg,	J2=    90.000 deg
};
P[1184]{
   GP1:
	UF : 1, UT : 1,		CONFIG : 'N U T, 0, 0, -1',
	X =  2339.940  mm,	Y =  -373.864  mm,	Z =   -66.156  mm,
	W =   -26.334 deg,	P =    14.915 deg,	R =   117.862 deg
   GP2:
	UF : 0, UT : 1,
	J1=    75.000 deg,	J2=    90.000 deg
};
P[1185]{
   GP1:
	UF : 1, UT : 1,		CONFIG : 'N U T, 0, 0, 0',
	X =  2342.079  mm,	Y =  -537.363  mm,	Z =   -66.325  mm,
	W =    18.926 deg,	P =    23.720 deg,	R =  -139.557 deg
   GP2:
	UF : 0, UT : 1,
	J1=    75.000 deg,	J2=    90.000 deg
};
P[1186]{
   GP1:
	UF : 1, UT : 1,		CONFIG : 'N U T, 0, 0, 0',
	X =  2367.990  mm,	Y =  -595.569  mm,	Z =   -71.145  mm,
	W =     7.550 deg,	P =    35.885 deg,	R =  -115.262 deg
   GP2:
	UF : 0, UT : 1,
	J1=    75.000 deg,	J2=    90.000 deg
};
P[1187]{
   GP1:
	UF : 1, UT : 1,		CONFIG : 'N U T, 0, 0, 0',
	X =  2418.261  mm,	Y =  -612.674  mm,	Z =   -84.509  mm,
	W =    26.080 deg,	P =    30.929 deg,	R =   -58.166 deg
   GP2:
	UF : 0, UT : 1,
	J1=    75.000 deg,	J2=    90.000 deg
};
P[1188]{
   GP1:
	UF : 1, UT : 1,		CONFIG : 'N U T, 0, 0, 0',
	X =  2506.701  mm,	Y =  -611.466  mm,	Z =  -107.718  mm,
	W =    38.274 deg,	P =    29.551 deg,	R =   -17.504 deg
   GP2:
	UF : 0, UT : 1,
	J1=    75.000 deg,	J2=    90.000 deg
};
P[1189]{
   GP1:
	UF : 1, UT : 1,		CONFIG : 'N U T, 0, 0, 0',
	X =  2543.054  mm,	Y =  -626.595  mm,	Z =  -116.227  mm,
	W =    27.942 deg,	P =    21.435 deg,	R =   -69.668 deg
   GP2:
	UF : 0, UT : 1,
	J1=    75.000 deg,	J2=    90.000 deg
};
P[1190]{
   GP1:
	UF : 1, UT : 1,		CONFIG : 'N U T, 0, 0, 0',
	X =  2560.144  mm,	Y =  -669.781  mm,	Z =  -121.378  mm,
	W =    25.909 deg,	P =    15.700 deg,	R =  -121.699 deg
   GP2:
	UF : 0, UT : 1,
	J1=    75.000 deg,	J2=    90.000 deg
};
P[1191]{
   GP1:
	UF : 1, UT : 1,		CONFIG : 'N U T, 0, 0, 0',
	X =  2545.732  mm,	Y = -1058.839  mm,	Z =  -115.894  mm,
	W =    28.324 deg,	P =   -10.379 deg,	R =   -74.774 deg
   GP2:
	UF : 0, UT : 1,
	J1=    75.000 deg,	J2=    90.000 deg
};
P[1192]{
   GP1:
	UF : 1, UT : 1,		CONFIG : 'N U T, 0, 0, 0',
	X =  2473.167  mm,	Y = -1064.660  mm,	Z =    -1.690  mm,
	W =    28.324 deg,	P =   -10.379 deg,	R =   -74.774 deg
   GP2:
	UF : 0, UT : 1,
	J1=    75.000 deg,	J2=    90.000 deg
};
P[1193]{
   GP1:
	UF : 1, UT : 1,		CONFIG : 'N U T, 0, 0, 0',
	X =  2362.332  mm,	Y =  -948.704  mm,	Z =   -46.458  mm,
	W =     1.961 deg,	P =    -3.226 deg,	R =   -23.425 deg
   GP2:
	UF : 0, UT : 1,
	J1=    75.000 deg,	J2=    90.000 deg
};
P[1194]{
   GP1:
	UF : 1, UT : 1,		CONFIG : 'N U T, 0, 0, 0',
	X =  2400.361  mm,	Y = -1187.577  mm,	Z =     9.775  mm,
	W =   -23.326 deg,	P =   -26.866 deg,	R =    43.658 deg
   GP2:
	UF : 0, UT : 1,
	J1=    75.000 deg,	J2=    90.000 deg
};
P[1195]{
   GP1:
	UF : 1, UT : 1,		CONFIG : 'N U T, 0, 0, 0',
	X =  2405.778  mm,	Y = -1194.018  mm,	Z =   -81.151  mm,
	W =   -19.565 deg,	P =   -23.197 deg,	R =    42.067 deg
   GP2:
	UF : 0, UT : 1,
	J1=    75.000 deg,	J2=    90.000 deg
};
P[1196]{
   GP1:
	UF : 1, UT : 1,		CONFIG : 'N U T, 0, 0, 0',
	X =  2406.332  mm,	Y = -1178.229  mm,	Z =   -80.540  mm,
	W =   -19.573 deg,	P =   -23.200 deg,	R =    42.068 deg
   GP2:
	UF : 0, UT : 1,
	J1=    75.000 deg,	J2=    90.000 deg
};
P[1197]{
   GP1:
	UF : 1, UT : 1,		CONFIG : 'N U T, 0, 0, 0',
	X =  2412.348  mm,	Y = -1170.129  mm,	Z =   -84.284  mm,
	W =   -34.316 deg,	P =    -2.466 deg,	R =    34.366 deg
   GP2:
	UF : 0, UT : 1,
	J1=    75.000 deg,	J2=    90.000 deg
};
P[1198]{
   GP1:
	UF : 1, UT : 1,		CONFIG : 'N U T, 0, 0, 0',
	X =  2418.087  mm,	Y = -1169.925  mm,	Z =   -87.740  mm,
	W =   -40.398 deg,	P =    23.613 deg,	R =    19.582 deg
   GP2:
	UF : 0, UT : 1,
	J1=    75.000 deg,	J2=    90.000 deg
};
P[1199]{
   GP1:
	UF : 1, UT : 1,		CONFIG : 'N U T, 0, 0, 0',
	X =  2439.433  mm,	Y = -1169.404  mm,	Z =   -93.614  mm,
	W =   -44.348 deg,	P =    17.233 deg,	R =    12.103 deg
   GP2:
	UF : 0, UT : 1,
	J1=    75.000 deg,	J2=    90.000 deg
};
P[1200]{
   GP1:
	UF : 1, UT : 1,		CONFIG : 'N U T, 0, 0, 0',
	X =  2472.436  mm,	Y = -1163.119  mm,	Z =  -100.981  mm,
	W =   -40.740 deg,	P =    -7.860 deg,	R =    -3.014 deg
   GP2:
	UF : 0, UT : 1,
	J1=    75.000 deg,	J2=    90.000 deg
};
P[1201]{
   GP1:
	UF : 1, UT : 1,		CONFIG : 'N U T, 1, 0, 0',
	X =  2493.725  mm,	Y = -1147.093  mm,	Z =  -105.313  mm,
	W =   -32.159 deg,	P =   -17.167 deg,	R =     4.025 deg
   GP2:
	UF : 0, UT : 1,
	J1=    75.000 deg,	J2=    90.000 deg
};
P[1202]{
   GP1:
	UF : 1, UT : 1,		CONFIG : 'N U T, 0, 0, 0',
	X =  2528.380  mm,	Y = -1109.365  mm,	Z =  -111.576  mm,
	W =   -20.148 deg,	P =   -29.973 deg,	R =   -17.669 deg
   GP2:
	UF : 0, UT : 1,
	J1=    75.000 deg,	J2=    90.000 deg
};
P[1203]{
   GP1:
	UF : 1, UT : 1,		CONFIG : 'N U T, 0, 0, 0',
	X =  2541.479  mm,	Y = -1091.180  mm,	Z =  -116.139  mm,
	W =    -6.295 deg,	P =   -31.612 deg,	R =   -24.783 deg
   GP2:
	UF : 0, UT : 1,
	J1=    75.000 deg,	J2=    90.000 deg
};
P[1204]{
   GP1:
	UF : 1, UT : 1,		CONFIG : 'N U T, 0, 0, -1',
	X =  2547.416  mm,	Y = -1057.501  mm,	Z =  -115.092  mm,
	W =    15.380 deg,	P =   -26.138 deg,	R =   -37.572 deg
   GP2:
	UF : 0, UT : 1,
	J1=    75.000 deg,	J2=    90.000 deg
};
P[1205]{
   GP1:
	UF : 1, UT : 1,		CONFIG : 'N U T, 0, 0, -1',
	X =  2492.591  mm,	Y = -1065.447  mm,	Z =    35.797  mm,
	W =    23.408 deg,	P =   -26.810 deg,	R =   -46.665 deg
   GP2:
	UF : 0, UT : 1,
	J1=    75.000 deg,	J2=    90.000 deg
};
P[1206]{
   GP1:
	UF : 1, UT : 1,		CONFIG : 'N U T, 0, 0, 0',
	X =  2043.269  mm,	Y = -1065.447  mm,	Z =   330.490  mm,
	W =    32.980 deg,	P =   -22.407 deg,	R =   -62.157 deg
   GP2:
	UF : 0, UT : 1,
	J1=    75.000 deg,	J2=    90.000 deg
};
P[1207]{
   GP1:
	UF : 1, UT : 1,		CONFIG : 'N U T, 0, 0, 0',
	X =  1479.583  mm,	Y = -1194.231  mm,	Z =   574.890  mm,
	W =   -33.532 deg,	P =   -24.491 deg,	R =   -26.069 deg
   GP2:
	UF : 0, UT : 1,
	J1=    75.000 deg,	J2=    90.000 deg
};
P[1208]{
   GP1:
	UF : 1, UT : 1,		CONFIG : 'N U T, 0, 0, 0',
	X =   469.561  mm,	Y =  -952.347  mm,	Z =   800.940  mm,
	W =      .899 deg,	P =    43.704 deg,	R =    71.522 deg
   GP2:
	UF : 0, UT : 1,
	J1=    75.000 deg,	J2=    90.000 deg
};
P[1209]{
   GP1:
	UF : 1, UT : 1,		CONFIG : 'N U T, 0, 0, 0',
	X =   744.220  mm,	Y =   -16.340  mm,	Z =  1493.482  mm,
	W =   -28.142 deg,	P =    21.236 deg,	R =    52.683 deg
   GP2:
	UF : 0, UT : 1,
	J1=    75.000 deg,	J2=    90.000 deg
};
P[1210]{
   GP1:
	UF : 1, UT : 1,		CONFIG : 'N U T, 0, 0, -1',
	X =  1934.433  mm,	Y =    90.324  mm,	Z =  1230.829  mm,
	W =   -12.673 deg,	P =    53.769 deg,	R =   143.611 deg
   GP2:
	UF : 0, UT : 1,
	J1=    90.000 deg,	J2=    90.000 deg
};
P[1211]{
   GP1:
	UF : 1, UT : 1,		CONFIG : 'N U T, 0, 0, -1',
	X =  2057.927  mm,	Y =    81.682  mm,	Z =   950.884  mm,
	W =    -3.033 deg,	P =    45.239 deg,	R =   153.300 deg
   GP2:
	UF : 0, UT : 1,
	J1=    90.000 deg,	J2=    90.000 deg
};
P[1212]{
   GP1:
	UF : 1, UT : 1,		CONFIG : 'N U T, 0, 0, -1',
	X =  2083.640  mm,	Y =    86.644  mm,	Z =   862.948  mm,
	W =     1.298 deg,	P =    45.759 deg,	R =   158.564 deg
   GP2:
	UF : 0, UT : 1,
	J1=    90.000 deg,	J2=    90.000 deg
};
P[1213]{
   GP1:
	UF : 1, UT : 1,		CONFIG : 'N U T, 0, 0, 0',
	X =  2073.865  mm,	Y =   117.284  mm,	Z =   860.519  mm,
	W =      .310 deg,	P =    44.767 deg,	R =  -121.017 deg
   GP2:
	UF : 0, UT : 1,
	J1=    89.999 deg,	J2=    90.000 deg
};
P[1214]{
   GP1:
	UF : 1, UT : 1,		CONFIG : 'N U T, 0, 0, 0',
	X =  2045.233  mm,	Y =   108.429  mm,	Z =   860.562  mm,
	W =     -.389 deg,	P =    43.845 deg,	R =   -25.335 deg
   GP2:
	UF : 0, UT : 1,
	J1=    89.999 deg,	J2=    90.000 deg
};
P[1215]{
   GP1:
	UF : 1, UT : 1,		CONFIG : 'N U T, 0, 0, 0',
	X =  2036.350  mm,	Y =    83.994  mm,	Z =   859.905  mm,
	W =     1.047 deg,	P =    44.551 deg,	R =   -14.937 deg
   GP2:
	UF : 0, UT : 1,
	J1=    90.000 deg,	J2=    90.000 deg
};
P[1216]{
   GP1:
	UF : 1, UT : 1,		CONFIG : 'N U T, 0, 0, 0',
	X =  2055.114  mm,	Y =    60.217  mm,	Z =   860.665  mm,
	W =      .512 deg,	P =    44.278 deg,	R =    68.687 deg
   GP2:
	UF : 0, UT : 1,
	J1=    90.000 deg,	J2=    90.000 deg
};
P[1217]{
   GP1:
	UF : 1, UT : 1,		CONFIG : 'N U T, 0, 0, 0',
	X =  2078.847  mm,	Y =    70.017  mm,	Z =   861.215  mm,
	W =      .619 deg,	P =    44.302 deg,	R =   160.837 deg
   GP2:
	UF : 0, UT : 1,
	J1=    90.000 deg,	J2=    90.000 deg
};
P[1218]{
   GP1:
	UF : 1, UT : 1,		CONFIG : 'N U T, 0, 0, 0',
	X =  2082.523  mm,	Y =    87.765  mm,	Z =   862.591  mm,
	W =      .679 deg,	P =    43.176 deg,	R =   162.144 deg
   GP2:
	UF : 0, UT : 1,
	J1=    90.000 deg,	J2=    90.000 deg
};
P[1219]{
   GP1:
	UF : 1, UT : 1,		CONFIG : 'N U T, 0, 0, 0',
	X =  2030.342  mm,	Y =   104.719  mm,	Z =  1095.609  mm,
	W =     4.326 deg,	P =    44.835 deg,	R =   168.123 deg
   GP2:
	UF : 0, UT : 1,
	J1=    90.000 deg,	J2=    90.000 deg
};
P[1220]{
   GP1:
	UF : 1, UT : 1,		CONFIG : 'N U T, 0, 0, 0',
	X =  2094.412  mm,	Y =   192.682  mm,	Z =  1020.508  mm,
	W =    -6.392 deg,	P =    42.881 deg,	R =    76.256 deg
   GP2:
	UF : 0, UT : 1,
	J1=    90.000 deg,	J2=    90.000 deg
};
P[1221]{
   GP1:
	UF : 1, UT : 1,		CONFIG : 'N U T, 0, 0, 0',
	X =  2055.715  mm,	Y =   156.952  mm,	Z =   864.739  mm,
	W =    -6.514 deg,	P =    44.590 deg,	R =    80.754 deg
   GP2:
	UF : 1, UT : 1,
	J1=    90.000 deg,	J2=    90.000 deg
};
P[1222]{
   GP1:
	UF : 1, UT : 1,		CONFIG : 'N U T, 0, 0, 0',
	X =  2175.980  mm,	Y =   155.212  mm,	Z =   865.187  mm,
	W =    -6.519 deg,	P =    44.584 deg,	R =    80.731 deg
   GP2:
	UF : 1, UT : 1,
	J1=    89.999 deg,	J2=    90.000 deg
};
P[1223]{
   GP1:
	UF : 1, UT : 1,		CONFIG : 'N U T, 0, 0, 0',
	X =  2232.675  mm,	Y =   130.480  mm,	Z =   863.368  mm,
	W =   -10.502 deg,	P =    44.016 deg,	R =    36.787 deg
   GP2:
	UF : 1, UT : 1,
	J1=    90.000 deg,	J2=    90.000 deg
};
P[1224]{
   GP1:
	UF : 1, UT : 1,		CONFIG : 'N U T, 0, 0, 0',
	X =  2253.801  mm,	Y =    86.743  mm,	Z =   863.438  mm,
	W =    -2.340 deg,	P =    43.506 deg,	R =    13.475 deg
   GP2:
	UF : 1, UT : 1,
	J1=    90.000 deg,	J2=    90.000 deg
};
P[1225]{
   GP1:
	UF : 1, UT : 1,		CONFIG : 'N U T, 0, 0, 0',
	X =  2357.269  mm,	Y =   -59.957  mm,	Z =   863.784  mm,
	W =     -.575 deg,	P =    46.049 deg,	R =    47.558 deg
   GP2:
	UF : 1, UT : 1,
	J1=    90.000 deg,	J2=    90.000 deg
};
P[1226]{
   GP1:
	UF : 1, UT : 1,		CONFIG : 'N U T, 0, 0, 0',
	X =  2543.201  mm,	Y =  -101.314  mm,	Z =   862.640  mm,
	W =    -1.367 deg,	P =    45.764 deg,	R =    89.270 deg
   GP2:
	UF : 1, UT : 1,
	J1=    90.000 deg,	J2=    90.000 deg
};
P[1227]{
   GP1:
	UF : 1, UT : 1,		CONFIG : 'N U T, 0, 0, 0',
	X =  2595.248  mm,	Y =  -114.923  mm,	Z =   862.093  mm,
	W =    -1.659 deg,	P =    44.976 deg,	R =    61.762 deg
   GP2:
	UF : 1, UT : 1,
	J1=    90.000 deg,	J2=    90.000 deg
};
P[1228]{
   GP1:
	UF : 1, UT : 1,		CONFIG : 'N U T, 0, 0, 0',
	X =  2619.721  mm,	Y =  -142.767  mm,	Z =   859.844  mm,
	W =   -27.973 deg,	P =    36.809 deg,	R =     1.495 deg
   GP2:
	UF : 1, UT : 1,
	J1=    90.000 deg,	J2=    90.000 deg
};
P[1229]{
   GP1:
	UF : 1, UT : 1,		CONFIG : 'N U T, 0, 0, 0',
	X =  2638.228  mm,	Y =  -180.207  mm,	Z =   862.719  mm,
	W =   -32.750 deg,	P =    30.016 deg,	R =     -.323 deg
   GP2:
	UF : 1, UT : 1,
	J1=    90.000 deg,	J2=    90.000 deg
};
P[1230]{
   GP1:
	UF : 1, UT : 1,		CONFIG : 'N U T, 0, 0, 0',
	X =  2663.091  mm,	Y =  -180.825  mm,	Z =   940.140  mm,
	W =   -32.753 deg,	P =    30.014 deg,	R =    10.111 deg
   GP2:
	UF : 0, UT : 1,
	J1=    90.000 deg,	J2=    90.000 deg
};
P[1231]{
   GP1:
	UF : 1, UT : 1,		CONFIG : 'N U T, 0, 0, 0',
	X =  2759.539  mm,	Y =  -352.824  mm,	Z =   940.140  mm,
	W =   -15.637 deg,	P =    18.786 deg,	R =    -8.670 deg
   GP2:
	UF : 0, UT : 1,
	J1=    90.000 deg,	J2=    90.000 deg
};
P[1232]{
   GP1:
	UF : 1, UT : 1,		CONFIG : 'N U T, 0, 0, 0',
	X =  2635.602  mm,	Y =  -179.163  mm,	Z =   864.410  mm,
	W =    11.258 deg,	P =    42.042 deg,	R =    39.085 deg
   GP2:
	UF : 0, UT : 1,
	J1=    89.999 deg,	J2=    90.000 deg
};
P[1233]{
   GP1:
	UF : 1, UT : 1,		CONFIG : 'N U T, 0, 0, 0',
	X =  2691.727  mm,	Y =  -303.823  mm,	Z =   865.455  mm,
	W =   -17.500 deg,	P =    36.921 deg,	R =     3.260 deg
   GP2:
	UF : 0, UT : 1,
	J1=    90.000 deg,	J2=    90.000 deg
};
P[1234]{
   GP1:
	UF : 1, UT : 1,		CONFIG : 'N U T, 0, 0, 0',
	X =  2732.146  mm,	Y =  -395.302  mm,	Z =   866.339  mm,
	W =   -28.374 deg,	P =    29.568 deg,	R =   -14.268 deg
   GP2:
	UF : 0, UT : 1,
	J1=    90.000 deg,	J2=    90.000 deg
};
P[1235]{
   GP1:
	UF : 1, UT : 1,		CONFIG : 'N U T, 0, 0, 0',
	X =  2778.109  mm,	Y =  -501.542  mm,	Z =   866.897  mm,
	W =   -36.634 deg,	P =    24.840 deg,	R =   -20.519 deg
   GP2:
	UF : 0, UT : 1,
	J1=    90.000 deg,	J2=    90.000 deg
};
P[1236]{
   GP1:
	UF : 1, UT : 1,		CONFIG : 'N U T, 0, 0, 0',
	X =  2870.505  mm,	Y =  -705.231  mm,	Z =   869.783  mm,
	W =   -42.548 deg,	P =     8.667 deg,	R =   -13.898 deg
   GP2:
	UF : 0, UT : 1,
	J1=    90.000 deg,	J2=    90.000 deg
};
P[1237]{
   GP1:
	UF : 1, UT : 1,		CONFIG : 'N U T, 0, 0, 0',
	X =  2899.487  mm,	Y =  -557.469  mm,	Z =   905.131  mm,
	W =   -40.224 deg,	P =    17.491 deg,	R =     -.029 deg
   GP2:
	UF : 0, UT : 1,
	J1=    90.000 deg,	J2=    90.000 deg
};
P[1238]{
   GP1:
	UF : 1, UT : 1,		CONFIG : 'N U T, 0, 0, 0',
	X =  2352.487  mm,	Y =  -106.469  mm,	Z =   905.131  mm,
	W =   -40.224 deg,	P =    17.491 deg,	R =   -11.143 deg
   GP2:
	UF : 0, UT : 1,
	J1=    90.000 deg,	J2=    90.000 deg
};
P[1239]{
   GP1:
	UF : 1, UT : 1,		CONFIG : 'N U T, 0, 0, 0',
	X =  2349.711  mm,	Y =  -142.767  mm,	Z =   874.878  mm,
	W =   -41.895 deg,	P =    18.208 deg,	R =    -8.798 deg
   GP2:
	UF : 0, UT : 1,
	J1=    90.000 deg,	J2=    90.000 deg
};
P[1240]{
   GP1:
	UF : 1, UT : 1,		CONFIG : 'N U T, 0, 0, 0',
	X =  2283.153  mm,	Y =  -109.355  mm,	Z =   872.819  mm,
	W =   -41.895 deg,	P =    18.207 deg,	R =    -8.798 deg
   GP2:
	UF : 0, UT : 1,
	J1=    90.000 deg,	J2=    90.000 deg
};
P[1241]{
   GP1:
	UF : 1, UT : 1,		CONFIG : 'N U T, 0, 0, 0',
	X =  2352.487  mm,	Y =  -106.469  mm,	Z =  1005.131  mm,
	W =   -40.224 deg,	P =    17.491 deg,	R =   -11.143 deg
   GP2:
	UF : 0, UT : 1,
	J1=    90.000 deg,	J2=    90.000 deg
};
P[1242]{
   GP1:
	UF : 1, UT : 1,		CONFIG : 'N U T, 0, 0, 0',
	X =  2248.487  mm,	Y =  -183.468  mm,	Z =  1050.131  mm,
	W =    39.867 deg,	P =   -18.417 deg,	R =   -24.499 deg
   GP2:
	UF : 0, UT : 1,
	J1=    90.000 deg,	J2=    90.000 deg
};
P[1243]{
   GP1:
	UF : 1, UT : 1,		CONFIG : 'N U T, 0, 0, 0',
	X =  2271.850  mm,	Y =  -133.562  mm,	Z =   876.059  mm,
	W =    39.929 deg,	P =   -18.389 deg,	R =   -24.535 deg
   GP2:
	UF : 0, UT : 1,
	J1=    90.000 deg,	J2=    90.000 deg
};
P[1244]{
   GP1:
	UF : 1, UT : 1,		CONFIG : 'N U T, 0, 0, 0',
	X =  2336.492  mm,	Y =  -169.512  mm,	Z =   876.840  mm,
	W =    39.847 deg,	P =   -18.420 deg,	R =   -24.482 deg
   GP2:
	UF : 0, UT : 1,
	J1=    90.000 deg,	J2=    90.000 deg
};
P[1245]{
   GP1:
	UF : 1, UT : 1,		CONFIG : 'N U T, 0, 0, 0',
	X =  2294.069  mm,	Y =  -220.014  mm,	Z =   945.099  mm,
	W =    21.148 deg,	P =   -20.624 deg,	R =   -17.529 deg
   GP2:
	UF : 0, UT : 1,
	J1=    90.000 deg,	J2=    90.000 deg
};
P[1246]{
   GP1:
	UF : 1, UT : 1,		CONFIG : 'N U T, 0, 0, 0',
	X =  2338.975  mm,	Y =   -36.178  mm,	Z =   950.438  mm,
	W =    13.335 deg,	P =    -3.235 deg,	R =   -13.309 deg
   GP2:
	UF : 0, UT : 1,
	J1=    90.000 deg,	J2=    90.000 deg
};
P[1247]{
   GP1:
	UF : 1, UT : 1,		CONFIG : 'N U T, 0, 0, 0',
	X =  2423.667  mm,	Y =  -138.414  mm,	Z =   969.098  mm,
	W =   -11.026 deg,	P =    39.710 deg,	R =   -20.881 deg
   GP2:
	UF : 0, UT : 1,
	J1=    90.000 deg,	J2=    90.000 deg
};
P[1248]{
   GP1:
	UF : 1, UT : 1,		CONFIG : 'N U T, 0, 0, 0',
	X =  2350.374  mm,	Y =  -143.477  mm,	Z =   872.621  mm,
	W =   -11.026 deg,	P =    39.710 deg,	R =   -35.737 deg
   GP2:
	UF : 0, UT : 1,
	J1=    90.000 deg,	J2=    90.000 deg
};
P[1249]{
   GP1:
	UF : 1, UT : 1,		CONFIG : 'N U T, 0, 0, 0',
	X =  2336.524  mm,	Y =  -170.304  mm,	Z =   870.271  mm,
	W =   -11.026 deg,	P =    39.710 deg,	R =   -41.174 deg
   GP2:
	UF : 0, UT : 1,
	J1=    90.000 deg,	J2=    90.000 deg
};
P[1250]{
   GP1:
	UF : 1, UT : 1,		CONFIG : 'N U T, 0, 0, 0',
	X =  2377.004  mm,	Y =  -164.282  mm,	Z =   904.705  mm,
	W =    -8.727 deg,	P =    37.605 deg,	R =   -39.738 deg
   GP2:
	UF : 0, UT : 1,
	J1=    90.000 deg,	J2=    90.000 deg
};
P[1251]{
   GP1:
	UF : 1, UT : 1,		CONFIG : 'N U T, 0, 0, 0',
	X =  1434.139  mm,	Y =   -96.053  mm,	Z =  1044.378  mm,
	W =    35.942 deg,	P =   -29.145 deg,	R =   -48.109 deg
   GP2:
	UF : 0, UT : 1,
	J1=    90.000 deg,	J2=    90.000 deg
};
P[1252]{
   GP1:
	UF : 1, UT : 1,		CONFIG : 'N U T, 0, 0, 0',
	X =  1598.946  mm,	Y =   -68.636  mm,	Z =   872.853  mm,
	W =    35.973 deg,	P =   -29.108 deg,	R =   -48.121 deg
   GP2:
	UF : 0, UT : 1,
	J1=    90.000 deg,	J2=    90.000 deg
};
P[1253]{
   GP1:
	UF : 1, UT : 1,		CONFIG : 'N U T, 0, 0, 0',
	X =  1669.518  mm,	Y =  -570.275  mm,	Z =   870.406  mm,
	W =    39.081 deg,	P =   -25.372 deg,	R =   -55.573 deg
   GP2:
	UF : 0, UT : 1,
	J1=    89.994 deg,	J2=    90.001 deg
};
P[1254]{
   GP1:
	UF : 1, UT : 1,		CONFIG : 'N U T, 0, 0, 0',
	X =  1593.706  mm,	Y =  -518.344  mm,	Z =   947.328  mm,
	W =    43.928 deg,	P =   -20.046 deg,	R =   -74.854 deg
   GP2:
	UF : 0, UT : 1,
	J1=    90.000 deg,	J2=    90.000 deg
};
P[1255]{
   GP1:
	UF : 1, UT : 1,		CONFIG : 'N U T, 0, 0, 0',
	X =  1462.748  mm,	Y =  -105.245  mm,	Z =  1006.284  mm,
	W =    28.753 deg,	P =    19.512 deg,	R =   -64.352 deg
   GP2:
	UF : 0, UT : 1,
	J1=    90.000 deg,	J2=    90.000 deg
};
P[1256]{
   GP1:
	UF : 1, UT : 1,		CONFIG : 'N U T, 0, 0, 0',
	X =  1692.820  mm,	Y =   -70.036  mm,	Z =  1058.761  mm,
	W =    -3.706 deg,	P =    39.360 deg,	R =     3.645 deg
   GP2:
	UF : 0, UT : 1,
	J1=    90.000 deg,	J2=    90.000 deg
};
P[1257]{
   GP1:
	UF : 1, UT : 1,		CONFIG : 'N U T, 0, 0, 0',
	X =  1619.799  mm,	Y =   -64.713  mm,	Z =   867.956  mm,
	W =    -3.411 deg,	P =    44.793 deg,	R =     3.190 deg
   GP2:
	UF : 0, UT : 1,
	J1=    90.000 deg,	J2=    90.000 deg
};
P[1258]{
   GP1:
	UF : 1, UT : 1,		CONFIG : 'N U T, 0, 0, 0',
	X =  1684.212  mm,	Y =  -567.545  mm,	Z =   867.215  mm,
	W =   -43.326 deg,	P =    11.035 deg,	R =   -70.449 deg
   GP2:
	UF : 0, UT : 1,
	J1=    90.000 deg,	J2=    90.000 deg
};
P[1259]{
   GP1:
	UF : 1, UT : 1,		CONFIG : 'N U T, 0, 0, 0',
	X =  1864.754  mm,	Y =  -445.803  mm,	Z =  1023.931  mm,
	W =   -42.752 deg,	P =    -6.233 deg,	R =   -60.128 deg
   GP2:
	UF : 0, UT : 1,
	J1=    90.000 deg,	J2=    90.000 deg
};
P[1260]{
   GP1:
	UF : 1, UT : 1,		CONFIG : 'N U T, 0, 0, 0',
	X =  1320.451  mm,	Y =   130.918  mm,	Z =  1174.439  mm,
	W =     3.785 deg,	P =    35.875 deg,	R =      .609 deg
   GP2:
	UF : 0, UT : 1,
	J1=    90.000 deg,	J2=    90.000 deg
};
P[1261]{
   GP1:
	UF : 1, UT : 1,		CONFIG : 'N U T, 0, 0, 0',
	X =   733.679  mm,	Y =   695.989  mm,	Z =  1351.019  mm,
	W =    -8.561 deg,	P =    33.775 deg,	R =    -6.417 deg
   GP2:
	UF : 0, UT : 1,
	J1=    90.000 deg,	J2=    90.000 deg
};
P[1262]{
   GP1:
	UF : 1, UT : 1,		CONFIG : 'N U T, 0, 0, 0',
	X =  2464.094  mm,	Y =  1570.269  mm,	Z =  1287.636  mm,
	W =    34.631 deg,	P =   -20.439 deg,	R =   -45.641 deg
   GP2:
	UF : 0, UT : 1,
	J1=    90.000 deg,	J2=    80.000 deg
};
P[1263]{
   GP1:
	UF : 1, UT : 1,		CONFIG : 'N U T, 0, 0, 0',
	X =  2557.417  mm,	Y =  1604.019  mm,	Z =   806.571  mm,
	W =    36.017 deg,	P =   -29.586 deg,	R =   -62.799 deg
   GP2:
	UF : 0, UT : 1,
	J1=    90.000 deg,	J2=    80.000 deg
};
P[1264]{
   GP1:
	UF : 1, UT : 1,		CONFIG : 'N U T, 0, 0, 0',
	X =  2773.443  mm,	Y =  1511.018  mm,	Z =   657.571  mm,
	W =    36.017 deg,	P =   -29.586 deg,	R =   -64.860 deg
   GP2:
	UF : 0, UT : 1,
	J1=    90.000 deg,	J2=    80.000 deg
};
P[1265]{
   GP1:
	UF : 1, UT : 1,		CONFIG : 'N U T, 0, 0, 0',
	X =  2840.667  mm,	Y =  1483.617  mm,	Z =   630.242  mm,
	W =    25.513 deg,	P =   -45.644 deg,	R =   -57.230 deg
   GP2:
	UF : 0, UT : 1,
	J1=    89.999 deg,	J2=    80.000 deg
};
P[1266]{
   GP1:
	UF : 1, UT : 1,		CONFIG : 'N U T, 0, 0, 0',
	X =  2866.334  mm,	Y =  1471.210  mm,	Z =   617.974  mm,
	W =    18.532 deg,	P =   -48.178 deg,	R =   -50.594 deg
   GP2:
	UF : 1, UT : 1,
	J1=    89.999 deg,	J2=    80.000 deg
};
P[1267]{
   GP1:
	UF : 1, UT : 1,		CONFIG : 'N U T, 0, 0, 0',
	X =  2864.460  mm,	Y =  1519.376  mm,	Z =   611.684  mm,
	W =    24.186 deg,	P =   -44.120 deg,	R =   -50.049 deg
   GP2:
	UF : 1, UT : 1,
	J1=    89.999 deg,	J2=    80.000 deg
};
P[1268]{
   GP1:
	UF : 1, UT : 1,		CONFIG : 'N U T, 0, 0, 0',
	X =  2832.116  mm,	Y =  1569.535  mm,	Z =   601.273  mm,
	W =    43.449 deg,	P =   -15.770 deg,	R =   -35.488 deg
   GP2:
	UF : 1, UT : 1,
	J1=    89.998 deg,	J2=    80.000 deg
};
P[1269]{
   GP1:
	UF : 1, UT : 1,		CONFIG : 'N U T, 0, 0, 0',
	X =  2826.594  mm,	Y =  1571.600  mm,	Z =   602.538  mm,
	W =    43.341 deg,	P =   -14.676 deg,	R =   -32.052 deg
   GP2:
	UF : 1, UT : 1,
	J1=    89.998 deg,	J2=    80.000 deg
};
P[1270]{
   GP1:
	UF : 1, UT : 1,		CONFIG : 'N U T, 0, 0, 0',
	X =  2766.778  mm,	Y =  1608.487  mm,	Z =   593.034  mm,
	W =    41.229 deg,	P =   -17.227 deg,	R =   -22.582 deg
   GP2:
	UF : 1, UT : 1,
	J1=    89.998 deg,	J2=    80.000 deg
};
P[1271]{
   GP1:
	UF : 1, UT : 1,		CONFIG : 'N U T, 0, 0, 0',
	X =  2718.383  mm,	Y =  1553.514  mm,	Z =   671.141  mm,
	W =    41.229 deg,	P =   -17.227 deg,	R =   -22.582 deg
   GP2:
	UF : 0, UT : 1,
	J1=    89.999 deg,	J2=    80.000 deg
};
P[1272]{
   GP1:
	UF : 1, UT : 1,		CONFIG : 'N U T, 0, 0, 0',
	X =  2626.676  mm,	Y =  1696.319  mm,	Z =   707.935  mm,
	W =   -50.219 deg,	P =    -7.077 deg,	R =    46.580 deg
   GP2:
	UF : 0, UT : 1,
	J1=    90.000 deg,	J2=    80.000 deg
};
P[1273]{
   GP1:
	UF : 1, UT : 1,		CONFIG : 'N U T, 0, 0, 0',
	X =  2760.964  mm,	Y =  1613.249  mm,	Z =   593.325  mm,
	W =   -51.641 deg,	P =    -8.212 deg,	R =    56.621 deg
   GP2:
	UF : 0, UT : 1,
	J1=    90.000 deg,	J2=    80.000 deg
};
P[1274]{
   GP1:
	UF : 1, UT : 1,		CONFIG : 'N U T, 0, 0, 0',
	X =  2781.190  mm,	Y =  1643.143  mm,	Z =   588.718  mm,
	W =   -51.569 deg,	P =    -8.041 deg,	R =    56.416 deg
   GP2:
	UF : 0, UT : 1,
	J1=    89.999 deg,	J2=    80.000 deg
};
P[1275]{
   GP1:
	UF : 1, UT : 1,		CONFIG : 'N U T, 0, 0, 0',
	X =  2622.631  mm,	Y =  1694.272  mm,	Z =   692.651  mm,
	W =   -54.549 deg,	P =   -20.575 deg,	R =    64.434 deg
   GP2:
	UF : 0, UT : 1,
	J1=    90.000 deg,	J2=    80.000 deg
};
P[1276]{
   GP1:
	UF : 1, UT : 1,		CONFIG : 'N U T, 0, 0, 0',
	X =  1360.375  mm,	Y =   792.895  mm,	Z =  1738.194  mm,
	W =    28.012 deg,	P =   -23.444 deg,	R =   -31.919 deg
   GP2:
	UF : 0, UT : 1,
	J1=    90.000 deg,	J2=    90.000 deg
};
P[1277]{
   GP1:
	UF : 1, UT : 1,		CONFIG : 'N U B, 0, 0, 0',
	X =   357.498  mm,	Y =    -1.017  mm,	Z =  2424.525  mm,
	W =     -.020 deg,	P =   -39.994 deg,	R =      .020 deg
   GP2:
	UF : 1, UT : 1,
	J1=    90.000 deg,	J2=    90.000 deg
};
P[1278]{
   GP1:
	UF : 1, UT : 1,
	J1=      .005 deg,	J2=   -44.424 deg,	J3=    65.270 deg,
	J4=      .005 deg,	J5=   -70.270 deg,	J6=     -.002 deg
   GP2:
	UF : 0, UT : 1,
	J1=   -90.000 deg,	J2=    90.000 deg
};
P[1279]{
   GP1:
	UF : 1, UT : 1,		CONFIG : 'N U T, 0, 0, 0',
	X =   888.146  mm,	Y =  -602.894  mm,	Z =  1079.964  mm,
	W =   -52.537 deg,	P =    -3.928 deg,	R =    83.324 deg
   GP2:
	UF : 0, UT : 1,
	J1=   -90.000 deg,	J2=    90.000 deg
};
P[1280]{
   GP1:
	UF : 1, UT : 1,		CONFIG : 'N U T, 0, 0, 0',
	X =  1652.146  mm,	Y =  -630.465  mm,	Z =   945.277  mm,
	W =   -52.537 deg,	P =    -3.928 deg,	R =    60.644 deg
   GP2:
	UF : 0, UT : 1,
	J1=   -90.000 deg,	J2=    90.000 deg
};
P[1281]{
   GP1:
	UF : 1, UT : 1,		CONFIG : 'N U T, 0, 0, 0',
	X =  1699.504  mm,	Y =  -710.975  mm,	Z =   866.171  mm,
	W =   -44.826 deg,	P =    -4.593 deg,	R =    61.393 deg
   GP2:
	UF : 1, UT : 1,
	J1=   -90.000 deg,	J2=    90.000 deg
};
P[1282]{
   GP1:
	UF : 1, UT : 1,		CONFIG : 'N U T, 0, 0, 0',
	X =  1946.820  mm,	Y =  -153.040  mm,	Z =   864.296  mm,
	W =   -45.563 deg,	P =    -3.332 deg,	R =    73.092 deg
   GP2:
	UF : 1, UT : 1,
	J1=   -90.000 deg,	J2=    90.000 deg
};
P[1283]{
   GP1:
	UF : 1, UT : 1,		CONFIG : 'N U T, 0, 0, 0',
	X =  1883.955  mm,	Y =  -143.969  mm,	Z =   930.742  mm,
	W =   -64.247 deg,	P =    -5.308 deg,	R =    92.033 deg
   GP2:
	UF : 0, UT : 1,
	J1=   -90.000 deg,	J2=    90.000 deg
};
P[1284]{
   GP1:
	UF : 1, UT : 1,		CONFIG : 'N U T, 0, 0, 0',
	X =  1347.073  mm,	Y =  -315.837  mm,	Z =   930.742  mm,
	W =   -64.247 deg,	P =    -5.308 deg,	R =    92.033 deg
   GP2:
	UF : 0, UT : 1,
	J1=   -90.000 deg,	J2=    90.000 deg
};
P[1285]{
   GP1:
	UF : 1, UT : 1,		CONFIG : 'N U T, 0, 0, 0',
	X =  1098.250  mm,	Y =  -457.920  mm,	Z =   864.783  mm,
	W =     2.070 deg,	P =     1.344 deg,	R =    -3.885 deg
   GP2:
	UF : 0, UT : 1,
	J1=   -90.000 deg,	J2=    90.000 deg
};
P[1286]{
   GP1:
	UF : 1, UT : 1,		CONFIG : 'N U T, 0, 0, 0',
	X =  1195.812  mm,	Y =  -666.774  mm,	Z =   950.277  mm,
	W =    58.410 deg,	P =     1.273 deg,	R =   -88.963 deg
   GP2:
	UF : 0, UT : 1,
	J1=   -90.000 deg,	J2=    90.000 deg
};
P[1287]{
   GP1:
	UF : 1, UT : 1,		CONFIG : 'N U T, 0, 0, 0',
	X =  1657.098  mm,	Y =  -779.646  mm,	Z =   930.742  mm,
	W =    45.135 deg,	P =   -18.028 deg,	R =   -72.006 deg
   GP2:
	UF : 0, UT : 1,
	J1=   -90.000 deg,	J2=    90.000 deg
};
P[1288]{
   GP1:
	UF : 1, UT : 1,		CONFIG : 'N U T, 0, 0, 0',
	X =  1679.287  mm,	Y =  -776.679  mm,	Z =   865.950  mm,
	W =    41.524 deg,	P =   -20.127 deg,	R =   -75.069 deg
   GP2:
	UF : 1, UT : 1,
	J1=   -90.000 deg,	J2=    90.000 deg
};
P[1289]{
   GP1:
	UF : 1, UT : 1,		CONFIG : 'N U T, 0, 0, 0',
	X =  1681.888  mm,	Y =  -796.672  mm,	Z =   865.913  mm,
	W =    41.000 deg,	P =   -20.477 deg,	R =   -62.404 deg
   GP2:
	UF : 1, UT : 1,
	J1=   -89.999 deg,	J2=    90.000 deg
};
P[1290]{
   GP1:
	UF : 1, UT : 1,		CONFIG : 'N U T, 0, 0, 0',
	X =  1683.514  mm,	Y =  -803.958  mm,	Z =   865.960  mm,
	W =    47.530 deg,	P =   -19.101 deg,	R =   -59.677 deg
   GP2:
	UF : 1, UT : 1,
	J1=   -89.998 deg,	J2=    90.000 deg
};
P[1291]{
   GP1:
	UF : 1, UT : 1,		CONFIG : 'N U T, 0, 0, 0',
	X =  1886.256  mm,	Y = -1187.653  mm,	Z =   869.034  mm,
	W =    47.353 deg,	P =    -9.874 deg,	R =   -68.868 deg
   GP2:
	UF : 1, UT : 1,
	J1=   -90.000 deg,	J2=    90.000 deg
};
P[1292]{
   GP1:
	UF : 1, UT : 1,		CONFIG : 'N U T, 0, 0, 0',
	X =  1856.770  mm,	Y = -1198.746  mm,	Z =   906.359  mm,
	W =    47.317 deg,	P =    -9.906 deg,	R =   -68.856 deg
   GP2:
	UF : 0, UT : 1,
	J1=   -90.000 deg,	J2=    90.000 deg
};
P[1293]{
   GP1:
	UF : 1, UT : 1,		CONFIG : 'N U T, 0, 0, 0',
	X =  1298.711  mm,	Y = -1056.858  mm,	Z =   942.419  mm,
	W =    51.862 deg,	P =   -14.128 deg,	R =   -65.340 deg
   GP2:
	UF : 0, UT : 1,
	J1=   -90.000 deg,	J2=    90.000 deg
};
P[1294]{
   GP1:
	UF : 1, UT : 1,		CONFIG : 'N U T, 0, 0, 0',
	X =   765.670  mm,	Y =  -903.969  mm,	Z =   930.742  mm,
	W =    45.135 deg,	P =   -18.028 deg,	R =   -72.006 deg
   GP2:
	UF : 0, UT : 1,
	J1=   -90.000 deg,	J2=    90.000 deg
};
P[1295]{
   GP1:
	UF : 1, UT : 1,		CONFIG : 'N U B, 0, 0, 0',
	X =   357.017  mm,	Y =     -.146  mm,	Z =  2433.121  mm,
	W =     -.021 deg,	P =   -39.773 deg,	R =      .020 deg
   GP2:
	UF : 0, UT : 1,
	J1=   -90.000 deg,	J2=    90.000 deg
};
P[1296]{
   GP1:
	UF : 1, UT : 1,
	J1=    32.560 deg,	J2=   -60.491 deg,	J3=    15.402 deg,
	J4=   -23.409 deg,	J5=   -41.316 deg,	J6=    84.551 deg
   GP2:
	UF : 0, UT : 1,
	J1=   -90.000 deg,	J2=   -90.000 deg
};
P[1297]{
   GP1:
	UF : 1, UT : 1,		CONFIG : 'N U T, 0, 0, 0',
	X =  1672.185  mm,	Y =   771.955  mm,	Z =   922.028  mm,
	W =   -53.210 deg,	P =    -2.950 deg,	R =    86.737 deg
   GP2:
	UF : 0, UT : 1,
	J1=   -90.000 deg,	J2=   -90.000 deg
};
P[1298]{
   GP1:
	UF : 1, UT : 1,		CONFIG : 'N U T, 0, 0, 0',
	X =  1681.183  mm,	Y =   773.813  mm,	Z =   858.475  mm,
	W =   -45.334 deg,	P =    -4.733 deg,	R =    88.292 deg
   GP2:
	UF : 1, UT : 1,
	J1=   -90.000 deg,	J2=   -90.000 deg
};
P[1299]{
   GP1:
	UF : 1, UT : 1,		CONFIG : 'N U T, 0, 0, 0',
	X =  1679.934  mm,	Y =   786.841  mm,	Z =   860.137  mm,
	W =   -45.324 deg,	P =    -4.767 deg,	R =    78.189 deg
   GP2:
	UF : 1, UT : 1,
	J1=   -90.000 deg,	J2=   -90.000 deg
};
P[1300]{
   GP1:
	UF : 1, UT : 1,		CONFIG : 'N U T, 0, 0, 0',
	X =  1685.027  mm,	Y =   806.421  mm,	Z =   859.551  mm,
	W =   -45.270 deg,	P =    -4.781 deg,	R =    62.005 deg
   GP2:
	UF : 1, UT : 1,
	J1=   -90.000 deg,	J2=   -90.000 deg
};
P[1301]{
   GP1:
	UF : 1, UT : 1,		CONFIG : 'N U T, 0, 0, 0',
	X =  1890.044  mm,	Y =  1189.801  mm,	Z =   860.889  mm,
	W =   -41.233 deg,	P =   -19.884 deg,	R =    40.949 deg
   GP2:
	UF : 1, UT : 1,
	J1=   -90.000 deg,	J2=   -90.000 deg
};
P[1302]{
   GP1:
	UF : 1, UT : 1,		CONFIG : 'N U T, 0, 0, 0',
	X =  1717.649  mm,	Y =  1211.638  mm,	Z =   952.045  mm,
	W =   -46.336 deg,	P =   -33.058 deg,	R =    54.067 deg
   GP2:
	UF : 0, UT : 1,
	J1=   -90.000 deg,	J2=   -90.000 deg
};
P[1303]{
   GP1:
	UF : 1, UT : 1,		CONFIG : 'N U T, 0, 0, 0',
	X =   784.649  mm,	Y =  1085.924  mm,	Z =   952.045  mm,
	W =   -46.336 deg,	P =   -33.058 deg,	R =    48.624 deg
   GP2:
	UF : 0, UT : 1,
	J1=   -90.000 deg,	J2=   -90.000 deg
};
P[1304]{
   GP1:
	UF : 1, UT : 1,		CONFIG : 'N U B, 0, 0, 0',
	X =   357.017  mm,	Y =     -.147  mm,	Z =  2433.121  mm,
	W =     -.021 deg,	P =   -39.773 deg,	R =      .020 deg
   GP2:
	UF : 0, UT : 1,
	J1=   -90.000 deg,	J2=   -90.000 deg
};
P[1305]{
   GP1:
	UF : 1, UT : 1,		CONFIG : 'N U T, 0, 0, 0',
	X =   830.852  mm,	Y =  -483.273  mm,	Z =  1732.743  mm,
	W =   -19.284 deg,	P =     3.297 deg,	R =    -8.755 deg
   GP2:
	UF : 0, UT : 1,
	J1=    90.000 deg,	J2=   -90.000 deg
};
P[1306]{
   GP1:
	UF : 1, UT : 1,		CONFIG : 'N U T, 0, 0, 0',
	X =   767.197  mm,	Y =  -738.866  mm,	Z =  1347.110  mm,
	W =      .000 deg,	P =    43.936 deg,	R =      .007 deg
   GP2:
	UF : 0, UT : 1,
	J1=    90.000 deg,	J2=   -90.000 deg
};
P[1307]{
   GP1:
	UF : 1, UT : 1,		CONFIG : 'N U T, 0, 0, 0',
	X =  1858.198  mm,	Y =  -123.866  mm,	Z =    88.528  mm,
	W =   -43.304 deg,	P =     8.281 deg,	R =    89.437 deg
   GP2:
	UF : 0, UT : 1,
	J1=    90.000 deg,	J2=   -90.000 deg
};
P[1308]{
   GP1:
	UF : 1, UT : 1,		CONFIG : 'N U T, 0, 0, 0',
	X =  2026.261  mm,	Y =   -44.698  mm,	Z =   -36.323  mm,
	W =   -40.063 deg,	P =    24.150 deg,	R =   114.480 deg
   GP2:
	UF : 1, UT : 1,
	J1=    89.999 deg,	J2=   -90.000 deg
};
P[1309]{
   GP1:
	UF : 1, UT : 1,		CONFIG : 'N U T, 0, 0, 1',
	X =  2043.083  mm,	Y =   -18.215  mm,	Z =   -33.835  mm,
	W =   -48.094 deg,	P =    24.245 deg,	R =   137.754 deg
   GP2:
	UF : 1, UT : 1,
	J1=    89.999 deg,	J2=   -90.000 deg
};
P[1310]{
   GP1:
	UF : 1, UT : 1,		CONFIG : 'N U T, 0, 0, 0',
	X =  1932.512  mm,	Y =   -84.081  mm,	Z =   104.389  mm,
	W =   -43.304 deg,	P =     8.281 deg,	R =   116.653 deg
   GP2:
	UF : 0, UT : 1,
	J1=    90.000 deg,	J2=   -90.000 deg
};
P[1311]{
   GP1:
	UF : 1, UT : 1,		CONFIG : 'N U T, 0, 0, 0',
	X =  1733.857  mm,	Y =  -543.587  mm,	Z =   134.680  mm,
	W =   -12.508 deg,	P =    -9.562 deg,	R =    72.347 deg
   GP2:
	UF : 0, UT : 1,
	J1=    90.000 deg,	J2=   -90.000 deg
};
P[1312]{
   GP1:
	UF : 1, UT : 1,		CONFIG : 'N U T, 0, 0, 0',
	X =  1591.198  mm,	Y = -1120.865  mm,	Z =   261.396  mm,
	W =    43.884 deg,	P =    -2.387 deg,	R =     2.487 deg
   GP2:
	UF : 0, UT : 1,
	J1=    90.000 deg,	J2=   -90.000 deg
};
P[1313]{
   GP1:
	UF : 1, UT : 1,		CONFIG : 'N U T, 0, 0, 0',
	X =  2598.196  mm,	Y = -1016.866  mm,	Z =    71.110  mm,
	W =    43.884 deg,	P =    -2.387 deg,	R =     2.487 deg
   GP2:
	UF : 0, UT : 1,
	J1=    90.000 deg,	J2=   -90.000 deg
};
P[1314]{
   GP1:
	UF : 1, UT : 1,		CONFIG : 'N U T, 0, 0, 0',
	X =  2647.118  mm,	Y =  -923.440  mm,	Z =   -25.150  mm,
	W =    44.948 deg,	P =    -2.436 deg,	R =     2.435 deg
   GP2:
	UF : 1, UT : 1,
	J1=    89.999 deg,	J2=   -90.000 deg
};
P[1315]{
   GP1:
	UF : 1, UT : 1,		CONFIG : 'N U T, 0, 0, 0',
	X =  2675.601  mm,	Y =  -922.760  mm,	Z =   -23.875  mm,
	W =    44.955 deg,	P =    -2.433 deg,	R =     2.437 deg
   GP2:
	UF : 1, UT : 1,
	J1=    90.000 deg,	J2=   -90.000 deg
};
P[1316]{
   GP1:
	UF : 1, UT : 1,		CONFIG : 'N U T, 0, 0, 0',
	X =  2690.016  mm,	Y =  -919.083  mm,	Z =   -24.165  mm,
	W =    34.700 deg,	P =    -4.479 deg,	R =    17.698 deg
   GP2:
	UF : 1, UT : 1,
	J1=    90.000 deg,	J2=   -90.000 deg
};
P[1317]{
   GP1:
	UF : 1, UT : 1,		CONFIG : 'N U T, 0, 0, 0',
	X =  2696.339  mm,	Y =  -911.261  mm,	Z =   -24.996  mm,
	W =    16.193 deg,	P =     8.102 deg,	R =    28.025 deg
   GP2:
	UF : 1, UT : 1,
	J1=    89.999 deg,	J2=   -90.000 deg
};
P[1318]{
   GP1:
	UF : 1, UT : 1,		CONFIG : 'N U T, 0, 0, 0',
	X =  2653.897  mm,	Y =  -983.627  mm,	Z =    56.187  mm,
	W =    43.915 deg,	P =    11.001 deg,	R =   -22.994 deg
   GP2:
	UF : 0, UT : 1,
	J1=    90.000 deg,	J2=   -90.000 deg
};
P[1319]{
   GP1:
	UF : 1, UT : 1,		CONFIG : 'N U T, 0, 0, 0',
	X =  1897.525  mm,	Y = -1008.960  mm,	Z =   159.950  mm,
	W =    44.948 deg,	P =    -2.436 deg,	R =    -7.767 deg
   GP2:
	UF : 0, UT : 1,
	J1=    90.000 deg,	J2=   -90.000 deg
};
P[1320]{
   GP1:
	UF : 1, UT : 1,		CONFIG : 'N U T, 0, 0, 0',
	X =  1897.524  mm,	Y = -1008.961  mm,	Z =   242.951  mm,
	W =   -41.218 deg,	P =   -19.941 deg,	R =   -32.390 deg
   GP2:
	UF : 0, UT : 1,
	J1=    90.000 deg,	J2=   -90.000 deg
};
P[1321]{
   GP1:
	UF : 1, UT : 1,		CONFIG : 'N U T, 0, 0, 0',
	X =  2509.525  mm,	Y =  -803.961  mm,	Z =   173.665  mm,
	W =   -40.704 deg,	P =   -21.130 deg,	R =   -18.431 deg
   GP2:
	UF : 0, UT : 1,
